LIN {X 0,Y 410.534,Z 444.335,A -85,B 0,C 180,E1 -10511.019,E2 -10511.019} C_VEL
LIN {X 0,Y 410.459,Z 447.37,A -85,B 0,C 180,E1 -10512.291,E2 -10512.291} C_VEL
LIN {X 0,Y 412.843,Z 460.26,A -85,B 0,C 180,E1 -10512.809,E2 -10512.809} C_VEL
LIN {X 0,Y 414.455,Z 473.213,A -85,B 0,C 180,E1 -10513.499,E2 -10513.499} C_VEL
LIN {X 0,Y 414.8,Z 477.532,A -85,B 0,C 180,E1 -10513.766,E2 -10513.766} C_VEL
LIN {X 0,Y 413.981,Z 489.912,A -85,B 0,C 180,E1 -10514.618,E2 -10514.618} C_VEL
LIN {X 0,Y 413.13,Z 501.048,A -85,B 0,C 180,E1 -10515.595,E2 -10515.595} C_VEL
LIN {X 0,Y 412.456,Z 511.121,A -85,B 0,C 180,E1 -10516.702,E2 -10516.702} C_VEL
LIN {X 0,Y 411.795,Z 520.263,A -85,B 0,C 180,E1 -10517.933,E2 -10517.933} C_VEL
LIN {X 0,Y 411.029,Z 529.203,A -85,B 0,C 180,E1 -10519.409,E2 -10519.409} C_VEL
LIN {X 0,Y 410.57,Z 536.417,A -85,B 0,C 180,E1 -10520.89,E2 -10520.89} C_VEL
LIN {X 0,Y 410.293,Z 541.303,A -85,B 0,C 180,E1 -10522.124,E2 -10522.124} C_VEL
LIN {X 0,Y 410.077,Z 546.418,A -85,B 0,C 180,E1 -10523.731,E2 -10523.731} C_VEL
LIN {X 0,Y 410.023,Z 549.684,A -85,B 0,C 180,E1 -10525.084,E2 -10525.084} C_VEL
LIN {X 0,Y 409.937,Z 551.546,A -85,B 0,C 180,E1 -10526.068,E2 -10526.068} C_VEL
LIN {X 0,Y 409.997,Z 553.956,A -85,B 0,C 180,E1 -10528.036,E2 -10528.036} C_VEL
LIN {X 0,Y 409.956,Z 554.566,A -85,B 0,C 180,E1 -10529.018,E2 -10529.018} C_VEL
LIN {X 0,Y 409.948,Z 554.761,A -85,B 0,C 180,E1 -10530,E2 -10530} C_VEL
LIN {X 0,Y 409.999,Z 553.907,A -85,B 0,C 180,E1 -10531.965,E2 -10531.965} C_VEL
LIN {X 0,Y 409.946,Z 552.887,A -85,B 0,C 180,E1 -10532.948,E2 -10532.948} C_VEL
LIN {X 0,Y 409.938,Z 551.437,A -85,B 0,C 180,E1 -10533.933,E2 -10533.933} C_VEL
LIN {X 0,Y 410.023,Z 548.439,A -85,B 0,C 180,E1 -10535.41,E2 -10535.41} C_VEL
LIN {X 0,Y 410.166,Z 544.376,A -85,B 0,C 180,E1 -10536.889,E2 -10536.889} C_VEL
LIN {X 0,Y 410.467,Z 538.12,A -85,B 0,C 180,E1 -10538.617,E2 -10538.617} C_VEL
LIN {X 0,Y 410.893,Z 531.306,A -85,B 0,C 180,E1 -10540.097,E2 -10540.097} C_VEL
LIN {X 0,Y 411.324,Z 524.356,A -85,B 0,C 180,E1 -10541.332,E2 -10541.332} C_VEL
LIN {X 0,Y 411.998,Z 515.999,A -85,B 0,C 180,E1 -10542.562,E2 -10542.562} C_VEL
LIN {X 0,Y 412.657,Z 505.728,A -85,B 0,C 180,E1 -10543.794,E2 -10543.794} C_VEL
LIN {X 0,Y 413.456,Z 494.162,A -85,B 0,C 180,E1 -10544.898,E2 -10544.898} C_VEL
LIN {X 0,Y 414.251,Z 482.81,A -85,B 0,C 180,E1 -10545.751,E2 -10545.751} C_VEL
LIN {X 0,Y 414.417,Z 475.557,A -85,B 0,C 180,E1 -10546.197,E2 -10546.197} C_VEL
LIN {X 0,Y 412.714,Z 461.921,A -85,B 0,C 180,E1 -10546.926,E2 -10546.926} C_VEL
LIN {X 0,Y 410.687,Z 449.667,A -85,B 0,C 180,E1 -10547.409,E2 -10547.409} C_VEL
LIN {X 0,Y 410.428,Z 447.964,A -85,B 0,C 180,E1 -10547.469,E2 -10547.469} C_VEL
LIN {X 0,Y 410.774,Z 440.007,A -85,B 0,C 180,E1 -10551.057,E2 -10551.057} C_VEL
LIN {X 0,Y 411.056,Z 433.097,A -85,B 0,C 180,E1 -10554.226,E2 -10554.226} C_VEL
LIN {X 0,Y 411.471,Z 426.207,A -85,B 0,C 180,E1 -10557.462,E2 -10557.462} C_VEL
LIN {X 0,Y 411.896,Z 420.472,A -85,B 0,C 180,E1 -10560.222,E2 -10560.222} C_VEL
LIN {X 0,Y 412.375,Z 414.103,A -85,B 0,C 180,E1 -10563.374,E2 -10563.374} C_VEL
LIN {X 0,Y 412.666,Z 410.157,A -85,B 0,C 180,E1 -10565.384,E2 -10565.384} C_VEL
LIN {X 0,Y 412.285,Z 405.559,A -85,B 0,C 180,E1 -10567.856,E2 -10567.856} C_VEL
LIN {X 0,Y 411.558,Z 400.956,A -85,B 0,C 180,E1 -10570.46,E2 -10570.46} C_VEL
LIN {X 0,Y 411.242,Z 399.261,A -85,B 0,C 180,E1 -10571.557,E2 -10571.557} C_VEL
LIN {X 0,Y 411.177,Z 399.269,A -85,B 0,C 180,E1 -10575.51,E2 -10575.51} C_VEL
LIN {X 0,Y 411.165,Z 399.27,A -85,B 0,C 180,E1 -10578.772,E2 -10578.772} C_VEL
LIN {X 0,Y 411.194,Z 399.264,A -85,B 0,C 180,E1 -10582.026,E2 -10582.026} C_VEL
LIN {X 0,Y 411.207,Z 399.263,A -85,B 0,C 180,E1 -10585.666,E2 -10585.666} C_VEL
LIN {X 0,Y 411.19,Z 399.268,A -85,B 0,C 180,E1 -10589.152,E2 -10589.152} C_VEL
LIN {X 0,Y 411.26,Z 399.256,A -85,B 0,C 180,E1 -10592.522,E2 -10592.522} C_VEL
LIN {X 0,Y 411.228,Z 399.261,A -85,B 0,C 180,E1 -10595.785,E2 -10595.785} C_VEL
LIN {X 0,Y 411.197,Z 399.267,A -85,B 0,C 180,E1 -10598.966,E2 -10598.966} C_VEL
LIN {X 0,Y 411.253,Z 399.257,A -85,B 0,C 180,E1 -10602.085,E2 -10602.085} C_VEL
LIN {X 0,Y 411.26,Z 399.259,A -85,B 0,C 180,E1 -10605.147,E2 -10605.147} C_VEL
LIN {X 0,Y 411.285,Z 399.253,A -85,B 0,C 180,E1 -10608.167,E2 -10608.167} C_VEL
LIN {X 0,Y 411.483,Z 399.228,A -85,B 0,C 180,E1 -10612.147,E2 -10612.147} C_VEL
LIN {X 0,Y 411.475,Z 399.229,A -85,B 0,C 180,E1 -10614.118,E2 -10614.118} C_VEL
LIN {X 0,Y 411.511,Z 399.224,A -85,B 0,C 180,E1 -10618.042,E2 -10618.042} C_VEL
LIN {X 0,Y 411.64,Z 399.208,A -85,B 0,C 180,E1 -10620,E2 -10620} C_VEL
LIN {X 0,Y 411.458,Z 399.234,A -85,B 0,C 180,E1 -10622.937,E2 -10622.937} C_VEL
LIN {X 0,Y 411.461,Z 399.234,A -85,B 0,C 180,E1 -10626.867,E2 -10626.867} C_VEL
LIN {X 0,Y 411.355,Z 399.247,A -85,B 0,C 180,E1 -10628.845,E2 -10628.845} C_VEL
LIN {X 0,Y 411.284,Z 399.253,A -85,B 0,C 180,E1 -10631.833,E2 -10631.833} C_VEL
LIN {X 0,Y 411.26,Z 399.259,A -85,B 0,C 180,E1 -10634.853,E2 -10634.853} C_VEL
LIN {X 0,Y 411.253,Z 399.257,A -85,B 0,C 180,E1 -10637.915,E2 -10637.915} C_VEL
LIN {X 0,Y 411.197,Z 399.267,A -85,B 0,C 180,E1 -10641.034,E2 -10641.034} C_VEL
LIN {X 0,Y 411.227,Z 399.261,A -85,B 0,C 180,E1 -10644.215,E2 -10644.215} C_VEL
LIN {X 0,Y 411.259,Z 399.256,A -85,B 0,C 180,E1 -10647.478,E2 -10647.478} C_VEL
LIN {X 0,Y 411.19,Z 399.268,A -85,B 0,C 180,E1 -10650.848,E2 -10650.848} C_VEL
LIN {X 0,Y 411.207,Z 399.264,A -85,B 0,C 180,E1 -10654.333,E2 -10654.333} C_VEL
LIN {X 0,Y 411.194,Z 399.264,A -85,B 0,C 180,E1 -10657.974,E2 -10657.974} C_VEL
LIN {X 0,Y 411.164,Z 399.269,A -85,B 0,C 180,E1 -10661.228,E2 -10661.228} C_VEL
LIN {X 0,Y 411.176,Z 399.27,A -85,B 0,C 180,E1 -10664.49,E2 -10664.49} C_VEL
LIN {X 0,Y 411.178,Z 399.269,A -85,B 0,C 180,E1 -10668.195,E2 -10668.195} C_VEL
LIN {X 0,Y 411.221,Z 399.264,A -85,B 0,C 180,E1 -10670.776,E2 -10670.776} C_VEL
LIN {X 0,Y 411.201,Z 399.266,A -85,B 0,C 180,E1 -10674.471,E2 -10674.471} C_VEL
LIN {X 0,Y 411.209,Z 399.265,A -85,B 0,C 180,E1 -10676.873,E2 -10676.873} C_VEL
LIN {X 0,Y 411.235,Z 399.263,A -85,B 0,C 180,E1 -10680.644,E2 -10680.644} C_VEL
LIN {X 0,Y 411.24,Z 399.258,A -85,B 0,C 180,E1 -10683.619,E2 -10683.619} C_VEL
LIN {X 0,Y 411.205,Z 399.264,A -85,B 0,C 180,E1 -10686.852,E2 -10686.852} C_VEL
LIN {X 0,Y 411.217,Z 399.263,A -85,B 0,C 180,E1 -10690.05,E2 -10690.05} C_VEL
LIN {X 0,Y 411.265,Z 399.255,A -85,B 0,C 180,E1 -10693.131,E2 -10693.131} C_VEL
LIN {X 0,Y 411.308,Z 399.251,A -85,B 0,C 180,E1 -10696.896,E2 -10696.896} C_VEL
LIN {X 0,Y 411.294,Z 399.255,A -85,B 0,C 180,E1 -10700.161,E2 -10700.161} C_VEL
LIN {X 0,Y 411.463,Z 399.231,A -85,B 0,C 180,E1 -10703.133,E2 -10703.133} C_VEL
LIN {X 0,Y 411.311,Z 399.249,A -85,B 0,C 180,E1 -10705.099,E2 -10705.099} C_VEL
LIN {X 0,Y 411.513,Z 399.227,A -85,B 0,C 180,E1 -10708.042,E2 -10708.042} C_VEL
LIN {X 0,Y 411.642,Z 399.211,A -85,B 0,C 180,E1 -10710,E2 -10710} C_VEL
LIN {X 0,Y 411.467,Z 399.231,A -85,B 0,C 180,E1 -10712.937,E2 -10712.937} C_VEL
LIN {X 0,Y 411.425,Z 399.238,A -85,B 0,C 180,E1 -10715.882,E2 -10715.882} C_VEL
LIN {X 0,Y 411.055,Z 399.284,A -85,B 0,C 180,E1 -10718.851,E2 -10718.851} C_VEL
LIN {X 0,Y 410.931,Z 399.893,A -85,B 0,C 180,E1 -10719.847,E2 -10719.847} C_VEL
LIN {X 0,Y 410.765,Z 403.877,A -85,B 0,C 180,E1 -10723.219,E2 -10723.219} C_VEL
LIN {X 0,Y 410.587,Z 407.911,A -85,B 0,C 180,E1 -10726.554,E2 -10726.554} C_VEL
LIN {X 0,Y 410.492,Z 408.997,A -85,B 0,C 180,E1 -10727.431,E2 -10727.431} C_VEL
LIN {X 0,Y 409.759,Z 410.069,A -85,B 0,C 180,E1 -10728.236,E2 -10728.236} C_VEL
LIN {X 0,Y 406.821,Z 411.984,A -85,B 0,C 180,E1 -10729.538,E2 -10729.538} C_VEL
LIN {X 0,Y 404.358,Z 413.528,A -85,B 0,C 180,E1 -10730.59,E2 -10730.59} C_VEL
LIN {X 0,Y 403.295,Z 414.632,A -85,B 0,C 180,E1 -10731.405,E2 -10731.405} C_VEL
LIN {X 0,Y 403.204,Z 414.98,A -85,B 0,C 180,E1 -10731.683,E2 -10731.683} C_VEL
LIN {X 0,Y 403.126,Z 419.403,A -85,B 0,C 180,E1 -10735.224,E2 -10735.224} C_VEL
LIN {X 0,Y 403.12,Z 419.529,A -85,B 0,C 180,E1 -10735.323,E2 -10735.323} C_VEL
LIN {X 0,Y 406.742,Z 435.397,A -85,B 0,C 180,E1 -10736.073,E2 -10736.073} C_VEL
LIN {X 0,Y 408.218,Z 444.133,A -85,B 0,C 180,E1 -10736.591,E2 -10736.591} C_VEL
LIN {X 0,Y 407.522,Z 455.702,A -85,B 0,C 180,E1 -10737.333,E2 -10737.333} C_VEL
LIN {X 0,Y 406.846,Z 466.667,A -85,B 0,C 180,E1 -10738.238,E2 -10738.238} C_VEL
LIN {X 0,Y 406.077,Z 477.882,A -85,B 0,C 180,E1 -10739.411,E2 -10739.411} C_VEL
LIN {X 0,Y 405.377,Z 487.193,A -85,B 0,C 180,E1 -10740.615,E2 -10740.615} C_VEL
LIN {X 0,Y 404.747,Z 495.157,A -85,B 0,C 180,E1 -10741.866,E2 -10741.866} C_VEL
LIN {X 0,Y 404.142,Z 503.143,A -85,B 0,C 180,E1 -10743.414,E2 -10743.414} C_VEL
LIN {X 0,Y 403.603,Z 509.906,A -85,B 0,C 180,E1 -10745.073,E2 -10745.073} C_VEL
LIN {X 0,Y 403.245,Z 515.072,A -85,B 0,C 180,E1 -10746.706,E2 -10746.706} C_VEL
LIN {X 0,Y 403.02,Z 518.865,A -85,B 0,C 180,E1 -10748.305,E2 -10748.305} C_VEL
LIN {X 0,Y 402.771,Z 521.882,A -85,B 0,C 180,E1 -10750.211,E2 -10750.211} C_VEL
LIN {X 0,Y 402.72,Z 523.128,A -85,B 0,C 180,E1 -10751.54,E2 -10751.54} C_VEL
LIN {X 0,Y 402.728,Z 523.627,A -85,B 0,C 180,E1 -10752.889,E2 -10752.889} C_VEL
LIN {X 0,Y 402.74,Z 523.385,A -85,B 0,C 180,E1 -10754.318,E2 -10754.318} C_VEL
LIN {X 0,Y 402.808,Z 522.35,A -85,B 0,C 180,E1 -10755.741,E2 -10755.741} C_VEL
LIN {X 0,Y 402.952,Z 520.541,A -85,B 0,C 180,E1 -10757.14,E2 -10757.14} C_VEL
LIN {X 0,Y 403.182,Z 517.849,A -85,B 0,C 180,E1 -10758.55,E2 -10758.55} C_VEL
LIN {X 0,Y 403.438,Z 514.039,A -85,B 0,C 180,E1 -10760.039,E2 -10760.039} C_VEL
LIN {X 0,Y 403.834,Z 509.049,A -85,B 0,C 180,E1 -10761.548,E2 -10761.548} C_VEL
LIN {X 0,Y 404.367,Z 502.647,A -85,B 0,C 180,E1 -10763.08,E2 -10763.08} C_VEL
LIN {X 0,Y 405.072,Z 494.485,A -85,B 0,C 180,E1 -10764.631,E2 -10764.631} C_VEL
LIN {X 0,Y 405.853,Z 485.639,A -85,B 0,C 180,E1 -10765.988,E2 -10765.988} C_VEL
LIN {X 0,Y 406.63,Z 476.25,A -85,B 0,C 180,E1 -10767.162,E2 -10767.162} C_VEL
LIN {X 0,Y 407.461,Z 465.3,A -85,B 0,C 180,E1 -10768.259,E2 -10768.259} C_VEL
LIN {X 0,Y 408.228,Z 453.199,A -85,B 0,C 180,E1 -10769.22,E2 -10769.22} C_VEL
LIN {X 0,Y 408.72,Z 443.775,A -85,B 0,C 180,E1 -10769.804,E2 -10769.804} C_VEL
LIN {X 0,Y 406.173,Z 431.616,A -85,B 0,C 180,E1 -10770.537,E2 -10770.537} C_VEL
LIN {X 0,Y 403.286,Z 420.513,A -85,B 0,C 180,E1 -10771.08,E2 -10771.08} C_VEL
LIN {X 0,Y 403.395,Z 416.813,A -85,B 0,C 180,E1 -10774.179,E2 -10774.179} C_VEL
LIN {X 0,Y 403.589,Z 412.981,A -85,B 0,C 180,E1 -10777.474,E2 -10777.474} C_VEL
LIN {X 0,Y 403.803,Z 409.322,A -85,B 0,C 180,E1 -10780.69,E2 -10780.69} C_VEL
LIN {X 0,Y 404.001,Z 405.837,A -85,B 0,C 180,E1 -10783.839,E2 -10783.839} C_VEL
LIN {X 0,Y 404.23,Z 402.512,A -85,B 0,C 180,E1 -10786.937,E2 -10786.937} C_VEL
LIN {X 0,Y 404.177,Z 400.432,A -85,B 0,C 180,E1 -10788.973,E2 -10788.973} C_VEL
LIN {X 0,Y 404.281,Z 400.133,A -85,B 0,C 180,E1 -10790.999,E2 -10790.999} C_VEL
LIN {X 0,Y 404.407,Z 400.113,A -85,B 0,C 180,E1 -10793.013,E2 -10793.013} C_VEL
LIN {X 0,Y 404.28,Z 400.129,A -85,B 0,C 180,E1 -10795.014,E2 -10795.014} C_VEL
LIN {X 0,Y 404.479,Z 400.105,A -85,B 0,C 180,E1 -10798.009,E2 -10798.009} C_VEL
LIN {X 0,Y 404.609,Z 400.087,A -85,B 0,C 180,E1 -10800,E2 -10800} C_VEL
LIN {X 0,Y 404.419,Z 400.112,A -85,B 0,C 180,E1 -10802.988,E2 -10802.988} C_VEL
LIN {X 0,Y 404.408,Z 400.113,A -85,B 0,C 180,E1 -10806.987,E2 -10806.987} C_VEL
LIN {X 0,Y 404.254,Z 400.132,A -85,B 0,C 180,E1 -10810.012,E2 -10810.012} C_VEL
LIN {X 0,Y 404.262,Z 400.131,A -85,B 0,C 180,E1 -10813.212,E2 -10813.212} C_VEL
LIN {X 0,Y 404.212,Z 400.137,A -85,B 0,C 180,E1 -10817.007,E2 -10817.007} C_VEL
LIN {X 0,Y 404.16,Z 400.143,A -85,B 0,C 180,E1 -10820.352,E2 -10820.352} C_VEL
LIN {X 0,Y 404.166,Z 400.141,A -85,B 0,C 180,E1 -10823.575,E2 -10823.575} C_VEL
LIN {X 0,Y 404.18,Z 400.141,A -85,B 0,C 180,E1 -10825.767,E2 -10825.767} C_VEL
LIN {X 0,Y 404.195,Z 400.139,A -85,B 0,C 180,E1 -10828,E2 -10828} C_VEL
LIN {X 0,Y 404.14,Z 400.146,A -85,B 0,C 180,E1 -10831.559,E2 -10831.559} C_VEL
LIN {X 0,Y 404.183,Z 400.143,A -85,B 0,C 180,E1 -10835.017,E2 -10835.017} C_VEL
LIN {X 0,Y 404.162,Z 400.145,A -85,B 0,C 180,E1 -10838.756,E2 -10838.756} C_VEL
LIN {X 0,Y 404.148,Z 400.147,A -85,B 0,C 180,E1 -10841.605,E2 -10841.605} C_VEL
LIN {X 0,Y 404.143,Z 400.147,A -85,B 0,C 180,E1 -10844.523,E2 -10844.523} C_VEL
LIN {X 0,Y 404.182,Z 400.333,A -85,B 0,C 180,E1 -10847.111,E2 -10847.111} C_VEL
LIN {X 0,Y 404.952,Z 404.545,A -85,B 0,C 180,E1 -10850.049,E2 -10850.049} C_VEL
LIN {X 0,Y 405.612,Z 408.992,A -85,B 0,C 180,E1 -10852.848,E2 -10852.848} C_VEL
LIN {X 0,Y 405.693,Z 412.911,A -85,B 0,C 180,E1 -10855.134,E2 -10855.134} C_VEL
LIN {X 0,Y 405.279,Z 417.229,A -85,B 0,C 180,E1 -10857.482,E2 -10857.482} C_VEL
LIN {X 0,Y 404.815,Z 422.492,A -85,B 0,C 180,E1 -10860.233,E2 -10860.233} C_VEL
LIN {X 0,Y 404.277,Z 429.369,A -85,B 0,C 180,E1 -10863.686,E2 -10863.686} C_VEL
LIN {X 0,Y 403.856,Z 437.27,A -85,B 0,C 180,E1 -10867.49,E2 -10867.49} C_VEL
LIN {X 0,Y 403.467,Z 444.131,A -85,B 0,C 180,E1 -10870.673,E2 -10870.673} C_VEL
LIN {X 0,Y 403.404,Z 447.055,A -85,B 0,C 180,E1 -10871.938,E2 -10871.938} C_VEL
LIN {X 0,Y 405.856,Z 459.934,A -85,B 0,C 180,E1 -10872.478,E2 -10872.478} C_VEL
LIN {X 0,Y 407.465,Z 472.667,A -85,B 0,C 180,E1 -10873.171,E2 -10873.171} C_VEL
LIN {X 0,Y 407.878,Z 479.72,A -85,B 0,C 180,E1 -10873.625,E2 -10873.625} C_VEL
LIN {X 0,Y 407.042,Z 491.446,A -85,B 0,C 180,E1 -10874.478,E2 -10874.478} C_VEL
LIN {X 0,Y 406.123,Z 502.634,A -85,B 0,C 180,E1 -10875.52,E2 -10875.52} C_VEL
LIN {X 0,Y 405.407,Z 513.072,A -85,B 0,C 180,E1 -10876.737,E2 -10876.737} C_VEL
LIN {X 0,Y 404.665,Z 521.747,A -85,B 0,C 180,E1 -10877.971,E2 -10877.971} C_VEL
LIN {X 0,Y 403.927,Z 530.331,A -85,B 0,C 180,E1 -10879.474,E2 -10879.474} C_VEL
LIN {X 0,Y 403.482,Z 537.235,A -85,B 0,C 180,E1 -10880.981,E2 -10880.981} C_VEL
LIN {X 0,Y 403.14,Z 542.775,A -85,B 0,C 180,E1 -10882.488,E2 -10882.488} C_VEL
LIN {X 0,Y 402.946,Z 547.124,A -85,B 0,C 180,E1 -10883.993,E2 -10883.993} C_VEL
LIN {X 0,Y 402.935,Z 549.437,A -85,B 0,C 180,E1 -10884.997,E2 -10884.997} C_VEL
LIN {X 0,Y 402.857,Z 551.29,A -85,B 0,C 180,E1 -10885.999,E2 -10885.999} C_VEL
LIN {X 0,Y 402.907,Z 553.694,A -85,B 0,C 180,E1 -10888.001,E2 -10888.001} C_VEL
LIN {X 0,Y 402.882,Z 554.301,A -85,B 0,C 180,E1 -10889.001,E2 -10889.001} C_VEL
LIN {X 0,Y 402.871,Z 554.486,A -85,B 0,C 180,E1 -10890,E2 -10890} C_VEL
LIN {X 0,Y 402.882,Z 554.249,A -85,B 0,C 180,E1 -10891,E2 -10891} C_VEL
LIN {X 0,Y 402.909,Z 553.622,A -85,B 0,C 180,E1 -10892,E2 -10892} C_VEL
LIN {X 0,Y 402.846,Z 552.596,A -85,B 0,C 180,E1 -10893,E2 -10893} C_VEL
LIN {X 0,Y 402.859,Z 551.134,A -85,B 0,C 180,E1 -10894.002,E2 -10894.002} C_VEL
LIN {X 0,Y 402.924,Z 548.124,A -85,B 0,C 180,E1 -10895.505,E2 -10895.505} C_VEL
LIN {X 0,Y 403.078,Z 544.046,A -85,B 0,C 180,E1 -10897.011,E2 -10897.011} C_VEL
LIN {X 0,Y 403.404,Z 537.772,A -85,B 0,C 180,E1 -10898.769,E2 -10898.769} C_VEL
LIN {X 0,Y 403.838,Z 530.939,A -85,B 0,C 180,E1 -10900.276,E2 -10900.276} C_VEL
LIN {X 0,Y 404.346,Z 523.971,A -85,B 0,C 180,E1 -10901.53,E2 -10901.53} C_VEL
LIN {X 0,Y 405.021,Z 515.589,A -85,B 0,C 180,E1 -10902.782,E2 -10902.782} C_VEL
LIN {X 0,Y 405.721,Z 505.059,A -85,B 0,C 180,E1 -10904.058,E2 -10904.058} C_VEL
LIN {X 0,Y 406.57,Z 493.673,A -85,B 0,C 180,E1 -10905.157,E2 -10905.157} C_VEL
LIN {X 0,Y 407.378,Z 482.257,A -85,B 0,C 180,E1 -10906.024,E2 -10906.024} C_VEL
LIN {X 0,Y 407.429,Z 475.56,A -85,B 0,C 180,E1 -10906.446,E2 -10906.446} C_VEL
LIN {X 0,Y 405.74,Z 462.081,A -85,B 0,C 180,E1 -10907.184,E2 -10907.184} C_VEL
LIN {X 0,Y 403.629,Z 449.579,A -85,B 0,C 180,E1 -10907.692,E2 -10907.692} C_VEL
LIN {X 0,Y 403.376,Z 447.773,A -85,B 0,C 180,E1 -10907.748,E2 -10907.748} C_VEL
LIN {X 0,Y 403.673,Z 440.877,A -85,B 0,C 180,E1 -10910.911,E2 -10910.911} C_VEL
LIN {X 0,Y 403.978,Z 433.991,A -85,B 0,C 180,E1 -10914.132,E2 -10914.132} C_VEL
LIN {X 0,Y 404.44,Z 426.747,A -85,B 0,C 180,E1 -10917.596,E2 -10917.596} C_VEL
LIN {X 0,Y 404.956,Z 420.241,A -85,B 0,C 180,E1 -10920.795,E2 -10920.795} C_VEL
LIN {X 0,Y 405.516,Z 413.356,A -85,B 0,C 180,E1 -10924.282,E2 -10924.282} C_VEL
LIN {X 0,Y 405.607,Z 409.937,A -85,B 0,C 180,E1 -10926.095,E2 -10926.095} C_VEL
LIN {X 0,Y 405.092,Z 405.284,A -85,B 0,C 180,E1 -10928.674,E2 -10928.674} C_VEL
LIN {X 0,Y 404.175,Z 400.141,A -85,B 0,C 180,E1 -10931.713,E2 -10931.713} C_VEL
LIN {X 0,Y 404.147,Z 400.145,A -85,B 0,C 180,E1 -10935.478,E2 -10935.478} C_VEL
LIN {X 0,Y 404.119,Z 400.146,A -85,B 0,C 180,E1 -10938.635,E2 -10938.635} C_VEL
LIN {X 0,Y 404.153,Z 400.144,A -85,B 0,C 180,E1 -10941.492,E2 -10941.492} C_VEL
LIN {X 0,Y 404.186,Z 400.14,A -85,B 0,C 180,E1 -10944.984,E2 -10944.984} C_VEL
LIN {X 0,Y 404.143,Z 400.143,A -85,B 0,C 180,E1 -10948.554,E2 -10948.554} C_VEL
LIN {X 0,Y 404.196,Z 400.135,A -85,B 0,C 180,E1 -10952,E2 -10952} C_VEL
LIN {X 0,Y 404.178,Z 400.141,A -85,B 0,C 180,E1 -10955.334,E2 -10955.334} C_VEL
LIN {X 0,Y 404.139,Z 400.144,A -85,B 0,C 180,E1 -10958.581,E2 -10958.581} C_VEL
LIN {X 0,Y 404.211,Z 400.134,A -85,B 0,C 180,E1 -10961.762,E2 -10961.762} C_VEL
LIN {X 0,Y 404.207,Z 400.138,A -85,B 0,C 180,E1 -10964.882,E2 -10964.882} C_VEL
LIN {X 0,Y 404.257,Z 400.128,A -85,B 0,C 180,E1 -10967.958,E2 -10967.958} C_VEL
LIN {X 0,Y 404.434,Z 400.106,A -85,B 0,C 180,E1 -10972.1,E2 -10972.1} C_VEL
LIN {X 0,Y 404.424,Z 400.107,A -85,B 0,C 180,E1 -10974.015,E2 -10974.015} C_VEL
LIN {X 0,Y 404.48,Z 400.1,A -85,B 0,C 180,E1 -10978.008,E2 -10978.008} C_VEL
LIN {X 0,Y 404.61,Z 400.084,A -85,B 0,C 180,E1 -10980,E2 -10980} C_VEL
LIN {X 0,Y 404.416,Z 400.111,A -85,B 0,C 180,E1 -10982.988,E2 -10982.988} C_VEL
LIN {X 0,Y 404.412,Z 400.113,A -85,B 0,C 180,E1 -10986.987,E2 -10986.987} C_VEL
LIN {X 0,Y 404.259,Z 400.128,A -85,B 0,C 180,E1 -10990.012,E2 -10990.012} C_VEL
LIN {X 0,Y 404.267,Z 400.129,A -85,B 0,C 180,E1 -10993.211,E2 -10993.211} C_VEL
LIN {X 0,Y 404.216,Z 400.136,A -85,B 0,C 180,E1 -10997.007,E2 -10997.007} C_VEL
LIN {X 0,Y 404.164,Z 400.141,A -85,B 0,C 180,E1 -11000.352,E2 -11000.352} C_VEL
LIN {X 0,Y 404.17,Z 400.139,A -85,B 0,C 180,E1 -11003.574,E2 -11003.574} C_VEL
LIN {X 0,Y 404.184,Z 400.136,A -85,B 0,C 180,E1 -11005.766,E2 -11005.766} C_VEL
LIN {X 0,Y 404.196,Z 400.136,A -85,B 0,C 180,E1 -11008,E2 -11008} C_VEL
LIN {X 0,Y 404.14,Z 400.142,A -85,B 0,C 180,E1 -11011.558,E2 -11011.558} C_VEL
LIN {X 0,Y 404.186,Z 400.139,A -85,B 0,C 180,E1 -11015.016,E2 -11015.016} C_VEL
LIN {X 0,Y 404.153,Z 400.144,A -85,B 0,C 180,E1 -11018.757,E2 -11018.757} C_VEL
LIN {X 0,Y 404.123,Z 400.145,A -85,B 0,C 180,E1 -11021.6,E2 -11021.6} C_VEL
LIN {X 0,Y 404.146,Z 400.145,A -85,B 0,C 180,E1 -11024.522,E2 -11024.522} C_VEL
LIN {X 0,Y 404.137,Z 400.143,A -85,B 0,C 180,E1 -11027.296,E2 -11027.296} C_VEL
LIN {X 0,Y 404.17,Z 400.139,A -85,B 0,C 180,E1 -11029.955,E2 -11029.955} C_VEL
LIN {X 0,Y 404.141,Z 400.144,A -85,B 0,C 180,E1 -11033.124,E2 -11033.124} C_VEL
LIN {X 0,Y 404.146,Z 400.144,A -85,B 0,C 180,E1 -11036.188,E2 -11036.188} C_VEL
LIN {X 0,Y 404.147,Z 400.142,A -85,B 0,C 180,E1 -11039.715,E2 -11039.715} C_VEL
LIN {X 0,Y 404.197,Z 400.136,A -85,B 0,C 180,E1 -11043.123,E2 -11043.123} C_VEL
LIN {X 0,Y 404.179,Z 400.138,A -85,B 0,C 180,E1 -11045.334,E2 -11045.334} C_VEL
LIN {X 0,Y 404.141,Z 400.146,A -85,B 0,C 180,E1 -11048.581,E2 -11048.581} C_VEL
LIN {X 0,Y 404.212,Z 400.134,A -85,B 0,C 180,E1 -11051.762,E2 -11051.762} C_VEL
LIN {X 0,Y 404.208,Z 400.136,A -85,B 0,C 180,E1 -11054.882,E2 -11054.882} C_VEL
LIN {X 0,Y 404.258,Z 400.13,A -85,B 0,C 180,E1 -11057.958,E2 -11057.958} C_VEL
LIN {X 0,Y 404.436,Z 400.108,A -85,B 0,C 180,E1 -11062.099,E2 -11062.099} C_VEL
LIN {X 0,Y 404.426,Z 400.11,A -85,B 0,C 180,E1 -11064.015,E2 -11064.015} C_VEL
LIN {X 0,Y 404.482,Z 400.102,A -85,B 0,C 180,E1 -11068.008,E2 -11068.008} C_VEL
LIN {X 0,Y 404.612,Z 400.087,A -85,B 0,C 180,E1 -11070,E2 -11070} C_VEL
LIN {X 0,Y 404.424,Z 400.108,A -85,B 0,C 180,E1 -11072.988,E2 -11072.988} C_VEL
LIN {X 0,Y 404.368,Z 400.117,A -85,B 0,C 180,E1 -11075.985,E2 -11075.985} C_VEL
LIN {X 0,Y 403.984,Z 400.165,A -85,B 0,C 180,E1 -11079.007,E2 -11079.007} C_VEL
LIN {X 0,Y 403.862,Z 400.935,A -85,B 0,C 180,E1 -11080.021,E2 -11080.021} C_VEL
LIN {X 0,Y 403.743,Z 404.494,A -85,B 0,C 180,E1 -11083.078,E2 -11083.078} C_VEL
LIN {X 0,Y 403.521,Z 408.816,A -85,B 0,C 180,E1 -11086.681,E2 -11086.681} C_VEL
LIN {X 0,Y 403.276,Z 413.4,A -85,B 0,C 180,E1 -11090.398,E2 -11090.398} C_VEL
LIN {X 0,Y 403.204,Z 414.98,A -85,B 0,C 180,E1 -11091.683,E2 -11091.683} C_VEL
LIN {X 0,Y 402.505,Z 415.721,A -85,B 0,C 180,E1 -11092.229,E2 -11092.229} C_VEL
LIN {X 0,Y 399.618,Z 417.05,A -85,B 0,C 180,E1 -11093.078,E2 -11093.078} C_VEL
LIN {X 0,Y 396.74,Z 418.386,A -85,B 0,C 180,E1 -11093.938,E2 -11093.938} C_VEL
LIN {X 0,Y 396.079,Z 419.139,A -85,B 0,C 180,E1 -11094.497,E2 -11094.497} C_VEL
LIN {X 0,Y 396.082,Z 419.813,A -85,B 0,C 180,E1 -11095.041,E2 -11095.041} C_VEL
LIN {X 0,Y 399.357,Z 434.224,A -85,B 0,C 180,E1 -11095.715,E2 -11095.715} C_VEL
LIN {X 0,Y 401.345,Z 445.277,A -85,B 0,C 180,E1 -11096.381,E2 -11096.381} C_VEL
LIN {X 0,Y 400.627,Z 456.648,A -85,B 0,C 180,E1 -11097.135,E2 -11097.135} C_VEL
LIN {X 0,Y 399.91,Z 467.292,A -85,B 0,C 180,E1 -11098.04,E2 -11098.04} C_VEL
LIN {X 0,Y 399.092,Z 478.629,A -85,B 0,C 180,E1 -11099.256,E2 -11099.256} C_VEL
LIN {X 0,Y 398.284,Z 488.808,A -85,B 0,C 180,E1 -11100.619,E2 -11100.619} C_VEL
LIN {X 0,Y 397.593,Z 497.229,A -85,B 0,C 180,E1 -11102.024,E2 -11102.024} C_VEL
LIN {X 0,Y 396.954,Z 505.221,A -85,B 0,C 180,E1 -11103.682,E2 -11103.682} C_VEL
LIN {X 0,Y 396.455,Z 511.588,A -85,B 0,C 180,E1 -11105.368,E2 -11105.368} C_VEL
LIN {X 0,Y 396.116,Z 516.57,A -85,B 0,C 180,E1 -11107.101,E2 -11107.101} C_VEL
LIN {X 0,Y 395.882,Z 519.848,A -85,B 0,C 180,E1 -11108.637,E2 -11108.637} C_VEL
LIN {X 0,Y 395.689,Z 522.173,A -85,B 0,C 180,E1 -11110.205,E2 -11110.205} C_VEL
LIN {X 0,Y 395.641,Z 523.508,A -85,B 0,C 180,E1 -11111.749,E2 -11111.749} C_VEL
LIN {X 0,Y 395.643,Z 523.932,A -85,B 0,C 180,E1 -11113.256,E2 -11113.256} C_VEL
LIN {X 0,Y 395.675,Z 523.104,A -85,B 0,C 180,E1 -11115.273,E2 -11115.273} C_VEL
LIN {X 0,Y 395.801,Z 521.553,A -85,B 0,C 180,E1 -11116.719,E2 -11116.719} C_VEL
LIN {X 0,Y 396.047,Z 519.129,A -85,B 0,C 180,E1 -11118.184,E2 -11118.184} C_VEL
LIN {X 0,Y 396.297,Z 515.685,A -85,B 0,C 180,E1 -11119.69,E2 -11119.69} C_VEL
LIN {X 0,Y 396.676,Z 511.092,A -85,B 0,C 180,E1 -11121.219,E2 -11121.219} C_VEL
LIN {X 0,Y 397.282,Z 504.061,A -85,B 0,C 180,E1 -11123.025,E2 -11123.025} C_VEL
LIN {X 0,Y 398.029,Z 495.82,A -85,B 0,C 180,E1 -11124.675,E2 -11124.675} C_VEL
LIN {X 0,Y 398.789,Z 487.425,A -85,B 0,C 180,E1 -11126.021,E2 -11126.021} C_VEL
LIN {X 0,Y 399.774,Z 476.785,A -85,B 0,C 180,E1 -11127.403,E2 -11127.403} C_VEL
LIN {X 0,Y 400.63,Z 466.306,A -85,B 0,C 180,E1 -11128.484,E2 -11128.484} C_VEL
LIN {X 0,Y 401.447,Z 454.004,A -85,B 0,C 180,E1 -11129.49,E2 -11129.49} C_VEL
LIN {X 0,Y 402.01,Z 445.718,A -85,B 0,C 180,E1 -11130.022,E2 -11130.022} C_VEL
LIN {X 0,Y 399.721,Z 434.053,A -85,B 0,C 180,E1 -11130.761,E2 -11130.761} C_VEL
LIN {X 0,Y 396.256,Z 420.786,A -85,B 0,C 180,E1 -11131.468,E2 -11131.468} C_VEL
LIN {X 0,Y 396.404,Z 416.875,A -85,B 0,C 180,E1 -11134.817,E2 -11134.817} C_VEL
LIN {X 0,Y 396.564,Z 413.064,A -85,B 0,C 180,E1 -11138.151,E2 -11138.151} C_VEL
LIN {X 0,Y 396.789,Z 409.453,A -85,B 0,C 180,E1 -11141.408,E2 -11141.408} C_VEL
LIN {X 0,Y 397.002,Z 406.008,A -85,B 0,C 180,E1 -11144.601,E2 -11144.601} C_VEL
LIN {X 0,Y 397.196,Z 402.737,A -85,B 0,C 180,E1 -11147.741,E2 -11147.741} C_VEL
LIN {X 0,Y 397.162,Z 401.019,A -85,B 0,C 180,E1 -11149.808,E2 -11149.808} C_VEL
LIN {X 0,Y 397.39,Z 400.989,A -85,B 0,C 180,E1 -11152.041,E2 -11152.041} C_VEL
LIN {X 0,Y 397.252,Z 401.004,A -85,B 0,C 180,E1 -11154.925,E2 -11154.925} C_VEL
LIN {X 0,Y 397.448,Z 400.981,A -85,B 0,C 180,E1 -11157.973,E2 -11157.973} C_VEL
LIN {X 0,Y 397.578,Z 400.963,A -85,B 0,C 180,E1 -11160,E2 -11160} C_VEL
LIN {X 0,Y 397.377,Z 400.989,A -85,B 0,C 180,E1 -11163.041,E2 -11163.041} C_VEL
LIN {X 0,Y 397.36,Z 400.991,A -85,B 0,C 180,E1 -11167.112,E2 -11167.112} C_VEL
LIN {X 0,Y 397.214,Z 401.009,A -85,B 0,C 180,E1 -11170.191,E2 -11170.191} C_VEL
LIN {X 0,Y 397.222,Z 401.007,A -85,B 0,C 180,E1 -11173.321,E2 -11173.321} C_VEL
LIN {X 0,Y 397.178,Z 401.013,A -85,B 0,C 180,E1 -11177.155,E2 -11177.155} C_VEL
LIN {X 0,Y 397.099,Z 401.022,A -85,B 0,C 180,E1 -11180.73,E2 -11180.73} C_VEL
LIN {X 0,Y 397.129,Z 401.016,A -85,B 0,C 180,E1 -11184.019,E2 -11184.019} C_VEL
LIN {X 0,Y 397.191,Z 401.011,A -85,B 0,C 180,E1 -11187.391,E2 -11187.391} C_VEL
LIN {X 0,Y 397.082,Z 401.026,A -85,B 0,C 180,E1 -11190.882,E2 -11190.882} C_VEL
LIN {X 0,Y 397.123,Z 401.02,A -85,B 0,C 180,E1 -11194.494,E2 -11194.494} C_VEL
LIN {X 0,Y 397.108,Z 401.024,A -85,B 0,C 180,E1 -11198.275,E2 -11198.275} C_VEL
LIN {X 0,Y 397.111,Z 401.023,A -85,B 0,C 180,E1 -11200.906,E2 -11200.906} C_VEL
LIN {X 0,Y 397.1,Z 401.024,A -85,B 0,C 180,E1 -11203.649,E2 -11203.649} C_VEL
LIN {X 0,Y 397.148,Z 401.216,A -85,B 0,C 180,E1 -11206.699,E2 -11206.699} C_VEL
LIN {X 0,Y 397.824,Z 405.035,A -85,B 0,C 180,E1 -11209.433,E2 -11209.433} C_VEL
LIN {X 0,Y 398.545,Z 409.725,A -85,B 0,C 180,E1 -11212.518,E2 -11212.518} C_VEL
LIN {X 0,Y 398.742,Z 412.909,A -85,B 0,C 180,E1 -11214.435,E2 -11214.435} C_VEL
LIN {X 0,Y 398.348,Z 417.163,A -85,B 0,C 180,E1 -11216.844,E2 -11216.844} C_VEL
LIN {X 0,Y 397.83,Z 422.941,A -85,B 0,C 180,E1 -11219.955,E2 -11219.955} C_VEL
LIN {X 0,Y 397.22,Z 430.344,A -85,B 0,C 180,E1 -11223.748,E2 -11223.748} C_VEL
LIN {X 0,Y 396.836,Z 437.105,A -85,B 0,C 180,E1 -11227.07,E2 -11227.07} C_VEL
LIN {X 0,Y 396.438,Z 443.913,A -85,B 0,C 180,E1 -11230.317,E2 -11230.317} C_VEL
LIN {X 0,Y 396.324,Z 446.553,A -85,B 0,C 180,E1 -11231.554,E2 -11231.554} C_VEL
LIN {X 0,Y 399.07,Z 460.698,A -85,B 0,C 180,E1 -11232.183,E2 -11232.183} C_VEL
LIN {X 0,Y 400.612,Z 473.302,A -85,B 0,C 180,E1 -11232.901,E2 -11232.901} C_VEL
LIN {X 0,Y 401.059,Z 479.993,A -85,B 0,C 180,E1 -11233.351,E2 -11233.351} C_VEL
LIN {X 0,Y 400.185,Z 491.419,A -85,B 0,C 180,E1 -11234.205,E2 -11234.205} C_VEL
LIN {X 0,Y 399.227,Z 502.535,A -85,B 0,C 180,E1 -11235.264,E2 -11235.264} C_VEL
LIN {X 0,Y 398.447,Z 513.138,A -85,B 0,C 180,E1 -11236.527,E2 -11236.527} C_VEL
LIN {X 0,Y 397.697,Z 521.593,A -85,B 0,C 180,E1 -11237.757,E2 -11237.757} C_VEL
LIN {X 0,Y 396.911,Z 530.146,A -85,B 0,C 180,E1 -11239.286,E2 -11239.286} C_VEL
LIN {X 0,Y 396.412,Z 537.035,A -85,B 0,C 180,E1 -11240.819,E2 -11240.819} C_VEL
LIN {X 0,Y 396.069,Z 542.562,A -85,B 0,C 180,E1 -11242.353,E2 -11242.353} C_VEL
LIN {X 0,Y 395.835,Z 547.638,A -85,B 0,C 180,E1 -11244.183,E2 -11244.183} C_VEL
LIN {X 0,Y 395.779,Z 551.044,A -85,B 0,C 180,E1 -11245.927,E2 -11245.927} C_VEL
LIN {X 0,Y 395.805,Z 553.435,A -85,B 0,C 180,E1 -11247.965,E2 -11247.965} C_VEL
LIN {X 0,Y 395.81,Z 554.038,A -85,B 0,C 180,E1 -11248.983,E2 -11248.983} C_VEL
LIN {X 0,Y 395.797,Z 554.21,A -85,B 0,C 180,E1 -11250,E2 -11250} C_VEL
LIN {X 0,Y 395.81,Z 553.968,A -85,B 0,C 180,E1 -11251.018,E2 -11251.018} C_VEL
LIN {X 0,Y 395.823,Z 553.335,A -85,B 0,C 180,E1 -11252.035,E2 -11252.035} C_VEL
LIN {X 0,Y 395.747,Z 552.303,A -85,B 0,C 180,E1 -11253.054,E2 -11253.054} C_VEL
LIN {X 0,Y 395.783,Z 550.828,A -85,B 0,C 180,E1 -11254.073,E2 -11254.073} C_VEL
LIN {X 0,Y 395.831,Z 547.295,A -85,B 0,C 180,E1 -11255.81,E2 -11255.81} C_VEL
LIN {X 0,Y 396.067,Z 542.077,A -85,B 0,C 180,E1 -11257.648,E2 -11257.648} C_VEL
LIN {X 0,Y 396.4,Z 536.393,A -85,B 0,C 180,E1 -11259.182,E2 -11259.182} C_VEL
LIN {X 0,Y 396.866,Z 529.255,A -85,B 0,C 180,E1 -11260.716,E2 -11260.716} C_VEL
LIN {X 0,Y 397.649,Z 520.366,A -85,B 0,C 180,E1 -11262.245,E2 -11262.245} C_VEL
LIN {X 0,Y 398.296,Z 511.648,A -85,B 0,C 180,E1 -11263.468,E2 -11263.468} C_VEL
LIN {X 0,Y 399.077,Z 501.195,A -85,B 0,C 180,E1 -11264.664,E2 -11264.664} C_VEL
LIN {X 0,Y 399.921,Z 490.058,A -85,B 0,C 180,E1 -11265.676,E2 -11265.676} C_VEL
LIN {X 0,Y 400.666,Z 478.604,A -85,B 0,C 180,E1 -11266.497,E2 -11266.497} C_VEL
LIN {X 0,Y 399.359,Z 466.306,A -85,B 0,C 180,E1 -11267.241,E2 -11267.241} C_VEL
LIN {X 0,Y 397.287,Z 453.084,A -85,B 0,C 180,E1 -11267.845,E2 -11267.845} C_VEL
LIN {X 0,Y 396.314,Z 447.476,A -85,B 0,C 180,E1 -11268.063,E2 -11268.063} C_VEL
LIN {X 0,Y 396.624,Z 440.591,A -85,B 0,C 180,E1 -11271.3,E2 -11271.3} C_VEL
LIN {X 0,Y 396.978,Z 433.715,A -85,B 0,C 180,E1 -11274.585,E2 -11274.585} C_VEL
LIN {X 0,Y 397.414,Z 427.049,A -85,B 0,C 180,E1 -11277.844,E2 -11277.844} C_VEL
LIN {X 0,Y 397.911,Z 421.135,A -85,B 0,C 180,E1 -11280.811,E2 -11280.811} C_VEL
LIN {X 0,Y 398.512,Z 414.28,A -85,B 0,C 180,E1 -11284.357,E2 -11284.357} C_VEL
LIN {X 0,Y 398.6,Z 411.586,A -85,B 0,C 180,E1 -11285.8,E2 -11285.8} C_VEL
LIN {X 0,Y 398.22,Z 407.393,A -85,B 0,C 180,E1 -11288.148,E2 -11288.148} C_VEL
LIN {X 0,Y 397.435,Z 402.797,A -85,B 0,C 180,E1 -11290.866,E2 -11290.866} C_VEL
LIN {X 0,Y 397.123,Z 401.02,A -85,B 0,C 180,E1 -11291.988,E2 -11291.988} C_VEL
LIN {X 0,Y 397.088,Z 401.025,A -85,B 0,C 180,E1 -11295.069,E2 -11295.069} C_VEL
LIN {X 0,Y 397.067,Z 401.024,A -85,B 0,C 180,E1 -11298.021,E2 -11298.021} C_VEL
LIN {X 0,Y 397.129,Z 401.019,A -85,B 0,C 180,E1 -11301.139,E2 -11301.139} C_VEL
LIN {X 0,Y 397.12,Z 401.017,A -85,B 0,C 180,E1 -11304.497,E2 -11304.497} C_VEL
LIN {X 0,Y 397.079,Z 401.022,A -85,B 0,C 180,E1 -11307.928,E2 -11307.928} C_VEL
LIN {X 0,Y 397.123,Z 401.019,A -85,B 0,C 180,E1 -11311.456,E2 -11311.456} C_VEL
LIN {X 0,Y 397.154,Z 401.013,A -85,B 0,C 180,E1 -11314.488,E2 -11314.488} C_VEL
LIN {X 0,Y 397.11,Z 401.022,A -85,B 0,C 180,E1 -11317.086,E2 -11317.086} C_VEL
LIN {X 0,Y 397.149,Z 401.013,A -85,B 0,C 180,E1 -11320.353,E2 -11320.353} C_VEL
LIN {X 0,Y 397.167,Z 401.012,A -85,B 0,C 180,E1 -11323.553,E2 -11323.553} C_VEL
LIN {X 0,Y 397.229,Z 401.005,A -85,B 0,C 180,E1 -11326.703,E2 -11326.703} C_VEL
LIN {X 0,Y 397.219,Z 401.004,A -85,B 0,C 180,E1 -11329.809,E2 -11329.809} C_VEL
LIN {X 0,Y 397.365,Z 400.99,A -85,B 0,C 180,E1 -11332.888,E2 -11332.888} C_VEL
LIN {X 0,Y 397.254,Z 401.004,A -85,B 0,C 180,E1 -11334.925,E2 -11334.925} C_VEL
LIN {X 0,Y 397.449,Z 400.975,A -85,B 0,C 180,E1 -11337.973,E2 -11337.973} C_VEL
LIN {X 0,Y 397.579,Z 400.96,A -85,B 0,C 180,E1 -11340,E2 -11340} C_VEL
LIN {X 0,Y 397.375,Z 400.988,A -85,B 0,C 180,E1 -11343.041,E2 -11343.041} C_VEL
LIN {X 0,Y 397.365,Z 400.99,A -85,B 0,C 180,E1 -11347.112,E2 -11347.112} C_VEL
LIN {X 0,Y 397.218,Z 401.005,A -85,B 0,C 180,E1 -11350.191,E2 -11350.191} C_VEL
LIN {X 0,Y 397.227,Z 401.005,A -85,B 0,C 180,E1 -11353.321,E2 -11353.321} C_VEL
LIN {X 0,Y 397.182,Z 401.012,A -85,B 0,C 180,E1 -11357.155,E2 -11357.155} C_VEL
LIN {X 0,Y 397.103,Z 401.023,A -85,B 0,C 180,E1 -11360.73,E2 -11360.73} C_VEL
LIN {X 0,Y 397.134,Z 401.015,A -85,B 0,C 180,E1 -11364.018,E2 -11364.018} C_VEL
LIN {X 0,Y 397.195,Z 401.008,A -85,B 0,C 180,E1 -11367.39,E2 -11367.39} C_VEL
LIN {X 0,Y 397.079,Z 401.026,A -85,B 0,C 180,E1 -11370.882,E2 -11370.882} C_VEL
LIN {X 0,Y 397.126,Z 401.019,A -85,B 0,C 180,E1 -11374.493,E2 -11374.493} C_VEL
LIN {X 0,Y 397.102,Z 401.021,A -85,B 0,C 180,E1 -11378.275,E2 -11378.275} C_VEL
LIN {X 0,Y 397.089,Z 401.023,A -85,B 0,C 180,E1 -11380.909,E2 -11380.909} C_VEL
LIN {X 0,Y 397.102,Z 401.018,A -85,B 0,C 180,E1 -11383.648,E2 -11383.648} C_VEL
LIN {X 0,Y 397.103,Z 401.023,A -85,B 0,C 180,E1 -11386.521,E2 -11386.521} C_VEL
LIN {X 0,Y 397.116,Z 401.021,A -85,B 0,C 180,E1 -11390.423,E2 -11390.423} C_VEL
LIN {X 0,Y 397.111,Z 401.021,A -85,B 0,C 180,E1 -11394.265,E2 -11394.265} C_VEL
LIN {X 0,Y 397.116,Z 401.021,A -85,B 0,C 180,E1 -11396.727,E2 -11396.727} C_VEL
LIN {X 0,Y 397.126,Z 401.019,A -85,B 0,C 180,E1 -11400.296,E2 -11400.296} C_VEL
LIN {X 0,Y 397.196,Z 401.011,A -85,B 0,C 180,E1 -11402.61,E2 -11402.61} C_VEL
LIN {X 0,Y 397.135,Z 401.017,A -85,B 0,C 180,E1 -11405.982,E2 -11405.982} C_VEL
LIN {X 0,Y 397.141,Z 401.015,A -85,B 0,C 180,E1 -11409.704,E2 -11409.704} C_VEL
LIN {X 0,Y 397.184,Z 401.01,A -85,B 0,C 180,E1 -11412.845,E2 -11412.845} C_VEL
LIN {X 0,Y 397.231,Z 401.005,A -85,B 0,C 180,E1 -11416.702,E2 -11416.702} C_VEL
LIN {X 0,Y 397.219,Z 401.005,A -85,B 0,C 180,E1 -11419.809,E2 -11419.809} C_VEL
LIN {X 0,Y 397.367,Z 400.987,A -85,B 0,C 180,E1 -11422.888,E2 -11422.888} C_VEL
LIN {X 0,Y 397.256,Z 401,A -85,B 0,C 180,E1 -11424.925,E2 -11424.925} C_VEL
LIN {X 0,Y 397.451,Z 400.978,A -85,B 0,C 180,E1 -11427.973,E2 -11427.973} C_VEL
LIN {X 0,Y 397.581,Z 400.963,A -85,B 0,C 180,E1 -11430,E2 -11430} C_VEL
LIN {X 0,Y 397.382,Z 400.984,A -85,B 0,C 180,E1 -11433.041,E2 -11433.041} C_VEL
LIN {X 0,Y 397.312,Z 400.996,A -85,B 0,C 180,E1 -11436.092,E2 -11436.092} C_VEL
LIN {X 0,Y 396.901,Z 401.047,A -85,B 0,C 180,E1 -11439.17,E2 -11439.17} C_VEL
LIN {X 0,Y 396.721,Z 404.365,A -85,B 0,C 180,E1 -11442.273,E2 -11442.273} C_VEL
LIN {X 0,Y 396.505,Z 408.062,A -85,B 0,C 180,E1 -11445.418,E2 -11445.418} C_VEL
LIN {X 0,Y 396.362,Z 410.603,A -85,B 0,C 180,E1 -11447.543,E2 -11447.543} C_VEL
LIN {X 0,Y 396.187,Z 414.546,A -85,B 0,C 180,E1 -11450.78,E2 -11450.78} C_VEL
LIN {X 0,Y 396.069,Z 418.632,A -85,B 0,C 180,E1 -11454.086,E2 -11454.086} C_VEL
LIN {X 0,Y 396.079,Z 419.139,A -85,B 0,C 180,E1 -11454.497,E2 -11454.497} C_VEL
LIN {X 0,Y 396.093,Z 420.439,A -85,B 0,C 180,E1 -11454.83,E2 -11454.83} C_VEL
LIN {X 0,Y 396.091,Z 423.426,A -85,B 0,C 180,E1 -11455.107,E2 -11455.107} C_VEL
LIN {X 0,Y 395.536,Z 437.759,A -85,B 0,C 180,E1 -11455.721,E2 -11455.721} C_VEL
LIN {X 0,Y 394.605,Z 445.721,A -85,B 0,C 180,E1 -11456.117,E2 -11456.117} C_VEL
LIN {X 0,Y 394.353,Z 448.303,A -85,B 0,C 180,E1 -11456.282,E2 -11456.282} C_VEL
LIN {X 0,Y 393.451,Z 461.138,A -85,B 0,C 180,E1 -11457.222,E2 -11457.222} C_VEL
LIN {X 0,Y 392.652,Z 472.587,A -85,B 0,C 180,E1 -11458.314,E2 -11458.314} C_VEL
LIN {X 0,Y 391.791,Z 482.971,A -85,B 0,C 180,E1 -11459.557,E2 -11459.557} C_VEL
LIN {X 0,Y 391.048,Z 492.078,A -85,B 0,C 180,E1 -11460.901,E2 -11460.901} C_VEL
LIN {X 0,Y 390.322,Z 500.4,A -85,B 0,C 180,E1 -11462.419,E2 -11462.419} C_VEL
LIN {X 0,Y 389.757,Z 507.277,A -85,B 0,C 180,E1 -11463.985,E2 -11463.985} C_VEL
LIN {X 0,Y 389.326,Z 513.164,A -85,B 0,C 180,E1 -11465.676,E2 -11465.676} C_VEL
LIN {X 0,Y 388.976,Z 517.625,A -85,B 0,C 180,E1 -11467.346,E2 -11467.346} C_VEL
LIN {X 0,Y 388.707,Z 521.229,A -85,B 0,C 180,E1 -11469.257,E2 -11469.257} C_VEL
LIN {X 0,Y 388.572,Z 522.938,A -85,B 0,C 180,E1 -11470.625,E2 -11470.625} C_VEL
LIN {X 0,Y 388.561,Z 523.966,A -85,B 0,C 180,E1 -11472.134,E2 -11472.134} C_VEL
LIN {X 0,Y 388.552,Z 524.158,A -85,B 0,C 180,E1 -11473.655,E2 -11473.655} C_VEL
LIN {X 0,Y 388.578,Z 523.528,A -85,B 0,C 180,E1 -11475.14,E2 -11475.14} C_VEL
LIN {X 0,Y 388.702,Z 522.116,A -85,B 0,C 180,E1 -11476.602,E2 -11476.602} C_VEL
LIN {X 0,Y 388.946,Z 519.902,A -85,B 0,C 180,E1 -11478.044,E2 -11478.044} C_VEL
LIN {X 0,Y 389.172,Z 516.913,A -85,B 0,C 180,E1 -11479.449,E2 -11479.449} C_VEL
LIN {X 0,Y 389.615,Z 511.949,A -85,B 0,C 180,E1 -11481.218,E2 -11481.218} C_VEL
LIN {X 0,Y 390.228,Z 505.288,A -85,B 0,C 180,E1 -11483.008,E2 -11483.008} C_VEL
LIN {X 0,Y 390.981,Z 497.342,A -85,B 0,C 180,E1 -11484.685,E2 -11484.685} C_VEL
LIN {X 0,Y 391.877,Z 488.119,A -85,B 0,C 180,E1 -11486.223,E2 -11486.223} C_VEL
LIN {X 0,Y 392.82,Z 478.304,A -85,B 0,C 180,E1 -11487.538,E2 -11487.538} C_VEL
LIN {X 0,Y 393.751,Z 467.773,A -85,B 0,C 180,E1 -11488.678,E2 -11488.678} C_VEL
LIN {X 0,Y 394.585,Z 456.513,A -85,B 0,C 180,E1 -11489.643,E2 -11489.643} C_VEL
LIN {X 0,Y 395.284,Z 447.003,A -85,B 0,C 180,E1 -11490.29,E2 -11490.29} C_VEL
LIN {X 0,Y 392.876,Z 435.006,A -85,B 0,C 180,E1 -11491.082,E2 -11491.082} C_VEL
LIN {X 0,Y 389.614,Z 422.987,A -85,B 0,C 180,E1 -11491.738,E2 -11491.738} C_VEL
LIN {X 0,Y 389.198,Z 421.097,A -85,B 0,C 180,E1 -11491.852,E2 -11491.852} C_VEL
LIN {X 0,Y 389.36,Z 416.944,A -85,B 0,C 180,E1 -11495.471,E2 -11495.471} C_VEL
LIN {X 0,Y 389.553,Z 413.181,A -85,B 0,C 180,E1 -11498.849,E2 -11498.849} C_VEL
LIN {X 0,Y 389.795,Z 409.596,A -85,B 0,C 180,E1 -11502.151,E2 -11502.151} C_VEL
LIN {X 0,Y 390.036,Z 406.195,A -85,B 0,C 180,E1 -11505.389,E2 -11505.389} C_VEL
LIN {X 0,Y 390.181,Z 404.03,A -85,B 0,C 180,E1 -11507.517,E2 -11507.517} C_VEL
LIN {X 0,Y 390.121,Z 401.981,A -85,B 0,C 180,E1 -11509.622,E2 -11509.622} C_VEL
LIN {X 0,Y 390.314,Z 401.869,A -85,B 0,C 180,E1 -11512.759,E2 -11512.759} C_VEL
LIN {X 0,Y 390.224,Z 401.879,A -85,B 0,C 180,E1 -11514.834,E2 -11514.834} C_VEL
LIN {X 0,Y 390.417,Z 401.857,A -85,B 0,C 180,E1 -11517.937,E2 -11517.937} C_VEL
LIN {X 0,Y 390.548,Z 401.839,A -85,B 0,C 180,E1 -11520,E2 -11520} C_VEL
LIN {X 0,Y 390.311,Z 401.869,A -85,B 0,C 180,E1 -11523.097,E2 -11523.097} C_VEL
LIN {X 0,Y 390.326,Z 401.867,A -85,B 0,C 180,E1 -11526.202,E2 -11526.202} C_VEL
LIN {X 0,Y 390.31,Z 401.868,A -85,B 0,C 180,E1 -11528.282,E2 -11528.282} C_VEL
LIN {X 0,Y 390.167,Z 401.886,A -85,B 0,C 180,E1 -11532.483,E2 -11532.483} C_VEL
LIN {X 0,Y 390.135,Z 401.889,A -85,B 0,C 180,E1 -11535.677,E2 -11535.677} C_VEL
LIN {X 0,Y 390.102,Z 401.894,A -85,B 0,C 180,E1 -11538.922,E2 -11538.922} C_VEL
LIN {X 0,Y 390.036,Z 401.902,A -85,B 0,C 180,E1 -11542.234,E2 -11542.234} C_VEL
LIN {X 0,Y 390.116,Z 401.893,A -85,B 0,C 180,E1 -11545.744,E2 -11545.744} C_VEL
LIN {X 0,Y 390.062,Z 401.899,A -85,B 0,C 180,E1 -11549.109,E2 -11549.109} C_VEL
LIN {X 0,Y 390.041,Z 401.902,A -85,B 0,C 180,E1 -11552.722,E2 -11552.722} C_VEL
LIN {X 0,Y 390.055,Z 401.902,A -85,B 0,C 180,E1 -11555.826,E2 -11555.826} C_VEL
LIN {X 0,Y 390.072,Z 401.901,A -85,B 0,C 180,E1 -11559.22,E2 -11559.22} C_VEL
LIN {X 0,Y 390.078,Z 401.899,A -85,B 0,C 180,E1 -11562.381,E2 -11562.381} C_VEL
LIN {X 0,Y 390.052,Z 401.915,A -85,B 0,C 180,E1 -11566.115,E2 -11566.115} C_VEL
LIN {X 0,Y 390.922,Z 406.744,A -85,B 0,C 180,E1 -11569.669,E2 -11569.669} C_VEL
LIN {X 0,Y 391.544,Z 410.815,A -85,B 0,C 180,E1 -11572.391,E2 -11572.391} C_VEL
LIN {X 0,Y 391.717,Z 415.005,A -85,B 0,C 180,E1 -11574.962,E2 -11574.962} C_VEL
LIN {X 0,Y 391.034,Z 421.435,A -85,B 0,C 180,E1 -11578.587,E2 -11578.587} C_VEL
LIN {X 0,Y 390.416,Z 428,A -85,B 0,C 180,E1 -11582.094,E2 -11582.094} C_VEL
LIN {X 0,Y 389.955,Z 434.676,A -85,B 0,C 180,E1 -11585.512,E2 -11585.512} C_VEL
LIN {X 0,Y 389.54,Z 441.449,A -85,B 0,C 180,E1 -11588.849,E2 -11588.849} C_VEL
LIN {X 0,Y 389.285,Z 446.264,A -85,B 0,C 180,E1 -11591.173,E2 -11591.173} C_VEL
LIN {X 0,Y 392.146,Z 460.469,A -85,B 0,C 180,E1 -11591.826,E2 -11591.826} C_VEL
LIN {X 0,Y 393.681,Z 472.866,A -85,B 0,C 180,E1 -11592.549,E2 -11592.549} C_VEL
LIN {X 0,Y 394.251,Z 480.263,A -85,B 0,C 180,E1 -11593.061,E2 -11593.061} C_VEL
LIN {X 0,Y 393.341,Z 491.47,A -85,B 0,C 180,E1 -11593.923,E2 -11593.923} C_VEL
LIN {X 0,Y 392.295,Z 503.211,A -85,B 0,C 180,E1 -11595.077,E2 -11595.077} C_VEL
LIN {X 0,Y 391.485,Z 513.21,A -85,B 0,C 180,E1 -11596.305,E2 -11596.305} C_VEL
LIN {X 0,Y 390.734,Z 521.456,A -85,B 0,C 180,E1 -11597.536,E2 -11597.536} C_VEL
LIN {X 0,Y 389.883,Z 529.963,A -85,B 0,C 180,E1 -11599.09,E2 -11599.09} C_VEL
LIN {X 0,Y 389.376,Z 536.837,A -85,B 0,C 180,E1 -11600.652,E2 -11600.652} C_VEL
LIN {X 0,Y 389.022,Z 542.35,A -85,B 0,C 180,E1 -11602.213,E2 -11602.213} C_VEL
LIN {X 0,Y 388.797,Z 546.8,A -85,B 0,C 180,E1 -11603.826,E2 -11603.826} C_VEL
LIN {X 0,Y 388.745,Z 548.974,A -85,B 0,C 180,E1 -11604.814,E2 -11604.814} C_VEL
LIN {X 0,Y 388.704,Z 550.8,A -85,B 0,C 180,E1 -11605.853,E2 -11605.853} C_VEL
LIN {X 0,Y 388.703,Z 553.178,A -85,B 0,C 180,E1 -11607.928,E2 -11607.928} C_VEL
LIN {X 0,Y 388.74,Z 553.775,A -85,B 0,C 180,E1 -11608.964,E2 -11608.964} C_VEL
LIN {X 0,Y 388.726,Z 553.933,A -85,B 0,C 180,E1 -11610,E2 -11610} C_VEL
LIN {X 0,Y 388.74,Z 553.684,A -85,B 0,C 180,E1 -11611.036,E2 -11611.036} C_VEL
LIN {X 0,Y 388.721,Z 553.042,A -85,B 0,C 180,E1 -11612.073,E2 -11612.073} C_VEL
LIN {X 0,Y 388.653,Z 552.002,A -85,B 0,C 180,E1 -11613.11,E2 -11613.11} C_VEL
LIN {X 0,Y 388.707,Z 550.51,A -85,B 0,C 180,E1 -11614.148,E2 -11614.148} C_VEL
LIN {X 0,Y 388.732,Z 547.335,A -85,B 0,C 180,E1 -11615.76,E2 -11615.76} C_VEL
LIN {X 0,Y 388.935,Z 543.348,A -85,B 0,C 180,E1 -11617.267,E2 -11617.267} C_VEL
LIN {X 0,Y 389.285,Z 537.029,A -85,B 0,C 180,E1 -11619.089,E2 -11619.089} C_VEL
LIN {X 0,Y 389.773,Z 530.145,A -85,B 0,C 180,E1 -11620.651,E2 -11620.651} C_VEL
LIN {X 0,Y 390.358,Z 523.12,A -85,B 0,C 180,E1 -11621.95,E2 -11621.95} C_VEL
LIN {X 0,Y 391.046,Z 514.663,A -85,B 0,C 180,E1 -11623.247,E2 -11623.247} C_VEL
LIN {X 0,Y 391.864,Z 504.226,A -85,B 0,C 180,E1 -11624.542,E2 -11624.542} C_VEL
LIN {X 0,Y 392.802,Z 492.517,A -85,B 0,C 180,E1 -11625.701,E2 -11625.701} C_VEL
LIN {X 0,Y 393.673,Z 480.871,A -85,B 0,C 180,E1 -11626.597,E2 -11626.597} C_VEL
LIN {X 0,Y 393.248,Z 473.724,A -85,B 0,C 180,E1 -11627.074,E2 -11627.074} C_VEL
LIN {X 0,Y 391.533,Z 460.419,A -85,B 0,C 180,E1 -11627.817,E2 -11627.817} C_VEL
LIN {X 0,Y 389.249,Z 447.29,A -85,B 0,C 180,E1 -11628.355,E2 -11628.355} C_VEL
LIN {X 0,Y 389.608,Z 440.304,A -85,B 0,C 180,E1 -11631.703,E2 -11631.703} C_VEL
LIN {X 0,Y 389.989,Z 433.449,A -85,B 0,C 180,E1 -11635.056,E2 -11635.056} C_VEL
LIN {X 0,Y 390.42,Z 427.346,A -85,B 0,C 180,E1 -11638.108,E2 -11638.108} C_VEL
LIN {X 0,Y 390.969,Z 420.888,A -85,B 0,C 180,E1 -11641.42,E2 -11641.42} C_VEL
LIN {X 0,Y 391.465,Z 415.384,A -85,B 0,C 180,E1 -11644.326,E2 -11644.326} C_VEL
LIN {X 0,Y 391.467,Z 410.599,A -85,B 0,C 180,E1 -11646.972,E2 -11646.972} C_VEL
LIN {X 0,Y 390.94,Z 406.498,A -85,B 0,C 180,E1 -11649.374,E2 -11649.374} C_VEL
LIN {X 0,Y 390.064,Z 401.9,A -85,B 0,C 180,E1 -11652.294,E2 -11652.294} C_VEL
LIN {X 0,Y 390.046,Z 401.902,A -85,B 0,C 180,E1 -11655.354,E2 -11655.354} C_VEL
LIN {X 0,Y 390.032,Z 401.899,A -85,B 0,C 180,E1 -11658.187,E2 -11658.187} C_VEL
LIN {X 0,Y 390.09,Z 401.895,A -85,B 0,C 180,E1 -11660.907,E2 -11660.907} C_VEL
LIN {X 0,Y 390.086,Z 401.895,A -85,B 0,C 180,E1 -11664.793,E2 -11664.793} C_VEL
LIN {X 0,Y 390.024,Z 401.901,A -85,B 0,C 180,E1 -11668.496,E2 -11668.496} C_VEL
LIN {X 0,Y 390.118,Z 401.888,A -85,B 0,C 180,E1 -11672.07,E2 -11672.07} C_VEL
LIN {X 0,Y 390.081,Z 401.896,A -85,B 0,C 180,E1 -11675.519,E2 -11675.519} C_VEL
LIN {X 0,Y 390.056,Z 401.9,A -85,B 0,C 180,E1 -11678.878,E2 -11678.878} C_VEL
LIN {X 0,Y 390.129,Z 401.887,A -85,B 0,C 180,E1 -11682.167,E2 -11682.167} C_VEL
LIN {X 0,Y 390.145,Z 401.888,A -85,B 0,C 180,E1 -11685.393,E2 -11685.393} C_VEL
LIN {X 0,Y 390.149,Z 401.887,A -85,B 0,C 180,E1 -11688.571,E2 -11688.571} C_VEL
LIN {X 0,Y 390.345,Z 401.86,A -85,B 0,C 180,E1 -11691.993,E2 -11691.993} C_VEL
LIN {X 0,Y 390.226,Z 401.879,A -85,B 0,C 180,E1 -11694.833,E2 -11694.833} C_VEL
LIN {X 0,Y 390.418,Z 401.851,A -85,B 0,C 180,E1 -11697.937,E2 -11697.937} C_VEL
LIN {X 0,Y 390.549,Z 401.835,A -85,B 0,C 180,E1 -11700,E2 -11700} C_VEL
LIN {X 0,Y 390.31,Z 401.869,A -85,B 0,C 180,E1 -11703.096,E2 -11703.096} C_VEL
LIN {X 0,Y 390.31,Z 401.864,A -85,B 0,C 180,E1 -11706.635,E2 -11706.635} C_VEL
LIN {X 0,Y 390.206,Z 401.88,A -85,B 0,C 180,E1 -11709.329,E2 -11709.329} C_VEL
LIN {X 0,Y 390.195,Z 401.88,A -85,B 0,C 180,E1 -11713.438,E2 -11713.438} C_VEL
LIN {X 0,Y 390.149,Z 401.887,A -85,B 0,C 180,E1 -11717.308,E2 -11717.308} C_VEL
LIN {X 0,Y 390.088,Z 401.895,A -85,B 0,C 180,E1 -11720.47,E2 -11720.47} C_VEL
LIN {X 0,Y 390.09,Z 401.893,A -85,B 0,C 180,E1 -11723.351,E2 -11723.351} C_VEL
LIN {X 0,Y 390.114,Z 401.893,A -85,B 0,C 180,E1 -11726.768,E2 -11726.768} C_VEL
LIN {X 0,Y 390.04,Z 401.901,A -85,B 0,C 180,E1 -11730.3,E2 -11730.3} C_VEL
LIN {X 0,Y 390.069,Z 401.895,A -85,B 0,C 180,E1 -11734.025,E2 -11734.025} C_VEL
LIN {X 0,Y 390.043,Z 401.897,A -85,B 0,C 180,E1 -11737.551,E2 -11737.551} C_VEL
LIN {X 0,Y 390.057,Z 401.9,A -85,B 0,C 180,E1 -11740.821,E2 -11740.821} C_VEL
LIN {X 0,Y 390.055,Z 401.896,A -85,B 0,C 180,E1 -11743.886,E2 -11743.886} C_VEL
LIN {X 0,Y 390.058,Z 401.9,A -85,B 0,C 180,E1 -11746.79,E2 -11746.79} C_VEL
LIN {X 0,Y 390.057,Z 401.895,A -85,B 0,C 180,E1 -11749.561,E2 -11749.561} C_VEL
LIN {X 0,Y 390.047,Z 401.901,A -85,B 0,C 180,E1 -11752.449,E2 -11752.449} C_VEL
LIN {X 0,Y 390.07,Z 401.895,A -85,B 0,C 180,E1 -11755.975,E2 -11755.975} C_VEL
LIN {X 0,Y 390.048,Z 401.898,A -85,B 0,C 180,E1 -11759.869,E2 -11759.869} C_VEL
LIN {X 0,Y 390.115,Z 401.889,A -85,B 0,C 180,E1 -11763.232,E2 -11763.232} C_VEL
LIN {X 0,Y 390.108,Z 401.893,A -85,B 0,C 180,E1 -11766.75,E2 -11766.75} C_VEL
LIN {X 0,Y 390.106,Z 401.892,A -85,B 0,C 180,E1 -11769.983,E2 -11769.983} C_VEL
LIN {X 0,Y 390.14,Z 401.885,A -85,B 0,C 180,E1 -11773.248,E2 -11773.248} C_VEL
LIN {X 0,Y 390.196,Z 401.882,A -85,B 0,C 180,E1 -11776.561,E2 -11776.561} C_VEL
LIN {X 0,Y 390.207,Z 401.881,A -85,B 0,C 180,E1 -11780.671,E2 -11780.671} C_VEL
LIN {X 0,Y 390.321,Z 401.866,A -85,B 0,C 180,E1 -11782.759,E2 -11782.759} C_VEL
LIN {X 0,Y 390.228,Z 401.876,A -85,B 0,C 180,E1 -11784.833,E2 -11784.833} C_VEL
LIN {X 0,Y 390.419,Z 401.854,A -85,B 0,C 180,E1 -11787.936,E2 -11787.936} C_VEL
LIN {X 0,Y 390.55,Z 401.838,A -85,B 0,C 180,E1 -11790,E2 -11790} C_VEL
LIN {X 0,Y 390.316,Z 401.864,A -85,B 0,C 180,E1 -11793.096,E2 -11793.096} C_VEL
LIN {X 0,Y 390.258,Z 401.875,A -85,B 0,C 180,E1 -11796.203,E2 -11796.203} C_VEL
LIN {X 0,Y 389.812,Z 401.93,A -85,B 0,C 180,E1 -11799.338,E2 -11799.338} C_VEL
LIN {X 0,Y 389.643,Z 406.12,A -85,B 0,C 180,E1 -11803.094,E2 -11803.094} C_VEL
LIN {X 0,Y 389.38,Z 410.631,A -85,B 0,C 180,E1 -11806.94,E2 -11806.94} C_VEL
LIN {X 0,Y 389.175,Z 414.392,A -85,B 0,C 180,E1 -11810.107,E2 -11810.107} C_VEL
LIN {X 0,Y 389.023,Z 418.449,A -85,B 0,C 180,E1 -11813.418,E2 -11813.418} C_VEL
LIN {X 0,Y 389.027,Z 420.133,A -85,B 0,C 180,E1 -11814.741,E2 -11814.741} C_VEL
LIN {X 0,Y 392.041,Z 433.29,A -85,B 0,C 180,E1 -11815.357,E2 -11815.357} C_VEL
LIN {X 0,Y 394.185,Z 443.997,A -85,B 0,C 180,E1 -11816.007,E2 -11816.007} C_VEL
LIN {X 0,Y 394.353,Z 448.303,A -85,B 0,C 180,E1 -11816.282,E2 -11816.282} C_VEL
LIN {X 0,Y 393.436,Z 451.956,A -85,B 0,C 180,E1 -11816.492,E2 -11816.492} C_VEL
LIN {X 0,Y 387.086,Z 463.096,A -85,B 0,C 180,E1 -11817.136,E2 -11817.136} C_VEL
LIN {X 0,Y 386.223,Z 466.406,A -85,B 0,C 180,E1 -11817.417,E2 -11817.417} C_VEL
LIN {X 0,Y 385.398,Z 477.236,A -85,B 0,C 180,E1 -11818.575,E2 -11818.575} C_VEL
LIN {X 0,Y 384.566,Z 486.956,A -85,B 0,C 180,E1 -11819.867,E2 -11819.867} C_VEL
LIN {X 0,Y 383.847,Z 494.877,A -85,B 0,C 180,E1 -11821.147,E2 -11821.147} C_VEL
LIN {X 0,Y 383.221,Z 501.715,A -85,B 0,C 180,E1 -11822.477,E2 -11822.477} C_VEL
LIN {X 0,Y 382.611,Z 509.088,A -85,B 0,C 180,E1 -11824.251,E2 -11824.251} C_VEL
LIN {X 0,Y 382.155,Z 514.818,A -85,B 0,C 180,E1 -11826.049,E2 -11826.049} C_VEL
LIN {X 0,Y 381.845,Z 518.77,A -85,B 0,C 180,E1 -11827.68,E2 -11827.68} C_VEL
LIN {X 0,Y 381.605,Z 521.662,A -85,B 0,C 180,E1 -11829.33,E2 -11829.33} C_VEL
LIN {X 0,Y 381.476,Z 523.493,A -85,B 0,C 180,E1 -11830.944,E2 -11830.944} C_VEL
LIN {X 0,Y 381.452,Z 524.453,A -85,B 0,C 180,E1 -11832.976,E2 -11832.976} C_VEL
LIN {X 0,Y 381.457,Z 524.226,A -85,B 0,C 180,E1 -11834.435,E2 -11834.435} C_VEL
LIN {X 0,Y 381.529,Z 523.229,A -85,B 0,C 180,E1 -11835.922,E2 -11835.922} C_VEL
LIN {X 0,Y 381.727,Z 521.4,A -85,B 0,C 180,E1 -11837.428,E2 -11837.428} C_VEL
LIN {X 0,Y 382.11,Z 517.528,A -85,B 0,C 180,E1 -11839.453,E2 -11839.453} C_VEL
LIN {X 0,Y 382.594,Z 512.386,A -85,B 0,C 180,E1 -11841.35,E2 -11841.35} C_VEL
LIN {X 0,Y 383.194,Z 506.428,A -85,B 0,C 180,E1 -11843.016,E2 -11843.016} C_VEL
LIN {X 0,Y 383.831,Z 500.03,A -85,B 0,C 180,E1 -11844.454,E2 -11844.454} C_VEL
LIN {X 0,Y 384.671,Z 491.673,A -85,B 0,C 180,E1 -11845.977,E2 -11845.977} C_VEL
LIN {X 0,Y 385.568,Z 483.084,A -85,B 0,C 180,E1 -11847.253,E2 -11847.253} C_VEL
LIN {X 0,Y 386.544,Z 473.124,A -85,B 0,C 180,E1 -11848.464,E2 -11848.464} C_VEL
LIN {X 0,Y 387.4,Z 462.872,A -85,B 0,C 180,E1 -11849.472,E2 -11849.472} C_VEL
LIN {X 0,Y 388.196,Z 451.737,A -85,B 0,C 180,E1 -11850.342,E2 -11850.342} C_VEL
LIN {X 0,Y 388.402,Z 447.034,A -85,B 0,C 180,E1 -11850.656,E2 -11850.656} C_VEL
LIN {X 0,Y 385.759,Z 434.606,A -85,B 0,C 180,E1 -11851.504,E2 -11851.504} C_VEL
LIN {X 0,Y 382.166,Z 421.41,A -85,B 0,C 180,E1 -11852.25,E2 -11852.25} C_VEL
LIN {X 0,Y 382.349,Z 417.036,A -85,B 0,C 180,E1 -11856.147,E2 -11856.147} C_VEL
LIN {X 0,Y 382.572,Z 413.288,A -85,B 0,C 180,E1 -11859.572,E2 -11859.572} C_VEL
LIN {X 0,Y 382.842,Z 409.757,A -85,B 0,C 180,E1 -11862.919,E2 -11862.919} C_VEL
LIN {X 0,Y 383.1,Z 406.127,A -85,B 0,C 180,E1 -11866.477,E2 -11866.477} C_VEL
LIN {X 0,Y 383.12,Z 403.273,A -85,B 0,C 180,E1 -11869.43,E2 -11869.43} C_VEL
LIN {X 0,Y 383.131,Z 402.768,A -85,B 0,C 180,E1 -11870.497,E2 -11870.497} C_VEL
LIN {X 0,Y 383.27,Z 402.747,A -85,B 0,C 180,E1 -11872.625,E2 -11872.625} C_VEL
LIN {X 0,Y 383.196,Z 402.755,A -85,B 0,C 180,E1 -11874.739,E2 -11874.739} C_VEL
LIN {X 0,Y 383.384,Z 402.733,A -85,B 0,C 180,E1 -11877.899,E2 -11877.899} C_VEL
LIN {X 0,Y 383.517,Z 402.715,A -85,B 0,C 180,E1 -11880,E2 -11880} C_VEL
LIN {X 0,Y 383.248,Z 402.748,A -85,B 0,C 180,E1 -11883.154,E2 -11883.154} C_VEL
LIN {X 0,Y 383.283,Z 402.744,A -85,B 0,C 180,E1 -11886.316,E2 -11886.316} C_VEL
LIN {X 0,Y 383.256,Z 402.747,A -85,B 0,C 180,E1 -11888.436,E2 -11888.436} C_VEL
LIN {X 0,Y 383.093,Z 402.767,A -85,B 0,C 180,E1 -11891.642,E2 -11891.642} C_VEL
LIN {X 0,Y 383.106,Z 402.765,A -85,B 0,C 180,E1 -11894.882,E2 -11894.882} C_VEL
LIN {X 0,Y 383.085,Z 402.769,A -85,B 0,C 180,E1 -11898.173,E2 -11898.173} C_VEL
LIN {X 0,Y 382.989,Z 402.78,A -85,B 0,C 180,E1 -11901.531,E2 -11901.531} C_VEL
LIN {X 0,Y 383.049,Z 402.773,A -85,B 0,C 180,E1 -11904.961,E2 -11904.961} C_VEL
LIN {X 0,Y 383.046,Z 402.773,A -85,B 0,C 180,E1 -11908.492,E2 -11908.492} C_VEL
LIN {X 0,Y 383.008,Z 402.779,A -85,B 0,C 180,E1 -11912.15,E2 -11912.15} C_VEL
LIN {X 0,Y 383.015,Z 402.778,A -85,B 0,C 180,E1 -11914.668,E2 -11914.668} C_VEL
LIN {X 0,Y 383.001,Z 402.782,A -85,B 0,C 180,E1 -11917.905,E2 -11917.905} C_VEL
LIN {X 0,Y 383.012,Z 402.78,A -85,B 0,C 180,E1 -11921.344,E2 -11921.344} C_VEL
LIN {X 0,Y 382.994,Z 402.78,A -85,B 0,C 180,E1 -11924.304,E2 -11924.304} C_VEL
LIN {X 0,Y 383.016,Z 402.974,A -85,B 0,C 180,E1 -11925.793,E2 -11925.793} C_VEL
LIN {X 0,Y 383.718,Z 406.822,A -85,B 0,C 180,E1 -11928.75,E2 -11928.75} C_VEL
LIN {X 0,Y 384.452,Z 411.225,A -85,B 0,C 180,E1 -11931.82,E2 -11931.82} C_VEL
LIN {X 0,Y 384.71,Z 414.979,A -85,B 0,C 180,E1 -11934.227,E2 -11934.227} C_VEL
LIN {X 0,Y 384.491,Z 418.147,A -85,B 0,C 180,E1 -11936.118,E2 -11936.118} C_VEL
LIN {X 0,Y 383.861,Z 423.912,A -85,B 0,C 180,E1 -11939.374,E2 -11939.374} C_VEL
LIN {X 0,Y 383.198,Z 431.2,A -85,B 0,C 180,E1 -11943.299,E2 -11943.299} C_VEL
LIN {X 0,Y 382.763,Z 437.683,A -85,B 0,C 180,E1 -11946.645,E2 -11946.645} C_VEL
LIN {X 0,Y 382.31,Z 444.704,A -85,B 0,C 180,E1 -11950.143,E2 -11950.143} C_VEL
LIN {X 0,Y 382.242,Z 446.13,A -85,B 0,C 180,E1 -11950.776,E2 -11950.776} C_VEL
LIN {X 0,Y 385.103,Z 459.775,A -85,B 0,C 180,E1 -11951.423,E2 -11951.423} C_VEL
LIN {X 0,Y 386.658,Z 471.364,A -85,B 0,C 180,E1 -11952.113,E2 -11952.113} C_VEL
LIN {X 0,Y 387.399,Z 480.49,A -85,B 0,C 180,E1 -11952.756,E2 -11952.756} C_VEL
LIN {X 0,Y 386.534,Z 491.511,A -85,B 0,C 180,E1 -11953.632,E2 -11953.632} C_VEL
LIN {X 0,Y 385.401,Z 503.193,A -85,B 0,C 180,E1 -11954.804,E2 -11954.804} C_VEL
LIN {X 0,Y 384.531,Z 513.32,A -85,B 0,C 180,E1 -11956.076,E2 -11956.076} C_VEL
LIN {X 0,Y 383.632,Z 522.874,A -85,B 0,C 180,E1 -11957.57,E2 -11957.57} C_VEL
LIN {X 0,Y 382.791,Z 531.067,A -85,B 0,C 180,E1 -11959.153,E2 -11959.153} C_VEL
LIN {X 0,Y 382.359,Z 536.661,A -85,B 0,C 180,E1 -11960.479,E2 -11960.479} C_VEL
LIN {X 0,Y 381.948,Z 542.148,A -85,B 0,C 180,E1 -11962.068,E2 -11962.068} C_VEL
LIN {X 0,Y 381.69,Z 546.978,A -85,B 0,C 180,E1 -11963.878,E2 -11963.878} C_VEL
LIN {X 0,Y 381.629,Z 550.556,A -85,B 0,C 180,E1 -11965.776,E2 -11965.776} C_VEL
LIN {X 0,Y 381.601,Z 552.922,A -85,B 0,C 180,E1 -11967.889,E2 -11967.889} C_VEL
LIN {X 0,Y 381.67,Z 553.511,A -85,B 0,C 180,E1 -11968.945,E2 -11968.945} C_VEL
LIN {X 0,Y 381.656,Z 553.657,A -85,B 0,C 180,E1 -11970,E2 -11970} C_VEL
LIN {X 0,Y 381.672,Z 553.4,A -85,B 0,C 180,E1 -11971.055,E2 -11971.055} C_VEL
LIN {X 0,Y 381.62,Z 552.749,A -85,B 0,C 180,E1 -11972.111,E2 -11972.111} C_VEL
LIN {X 0,Y 381.563,Z 551.699,A -85,B 0,C 180,E1 -11973.168,E2 -11973.168} C_VEL
LIN {X 0,Y 381.633,Z 550.193,A -85,B 0,C 180,E1 -11974.225,E2 -11974.225} C_VEL
LIN {X 0,Y 381.69,Z 546.398,A -85,B 0,C 180,E1 -11976.121,E2 -11976.121} C_VEL
LIN {X 0,Y 381.943,Z 541.362,A -85,B 0,C 180,E1 -11977.933,E2 -11977.933} C_VEL
LIN {X 0,Y 382.398,Z 534.507,A -85,B 0,C 180,E1 -11979.788,E2 -11979.788} C_VEL
LIN {X 0,Y 382.935,Z 527.05,A -85,B 0,C 180,E1 -11981.379,E2 -11981.379} C_VEL
LIN {X 0,Y 383.692,Z 519.464,A -85,B 0,C 180,E1 -11982.698,E2 -11982.698} C_VEL
LIN {X 0,Y 384.517,Z 509.949,A -85,B 0,C 180,E1 -11984.059,E2 -11984.059} C_VEL
LIN {X 0,Y 385.267,Z 500.082,A -85,B 0,C 180,E1 -11985.203,E2 -11985.203} C_VEL
LIN {X 0,Y 386.186,Z 488.827,A -85,B 0,C 180,E1 -11986.249,E2 -11986.249} C_VEL
LIN {X 0,Y 386.794,Z 478.945,A -85,B 0,C 180,E1 -11986.985,E2 -11986.985} C_VEL
LIN {X 0,Y 385.303,Z 465.964,A -85,B 0,C 180,E1 -11987.82,E2 -11987.82} C_VEL
LIN {X 0,Y 383.254,Z 453.251,A -85,B 0,C 180,E1 -11988.435,E2 -11988.435} C_VEL
LIN {X 0,Y 382.183,Z 446.999,A -85,B 0,C 180,E1 -11988.686,E2 -11988.686} C_VEL
LIN {X 0,Y 382.583,Z 440.004,A -85,B 0,C 180,E1 -11992.122,E2 -11992.122} C_VEL
LIN {X 0,Y 383.036,Z 432.336,A -85,B 0,C 180,E1 -11995.965,E2 -11995.965} C_VEL
LIN {X 0,Y 383.639,Z 425.187,A -85,B 0,C 180,E1 -11999.645,E2 -11999.645} C_VEL
LIN {X 0,Y 384.27,Z 418.347,A -85,B 0,C 180,E1 -12003.276,E2 -12003.276} C_VEL
LIN {X 0,Y 384.527,Z 413.782,A -85,B 0,C 180,E1 -12005.794,E2 -12005.794} C_VEL
LIN {X 0,Y 384.224,Z 409.733,A -85,B 0,C 180,E1 -12008.137,E2 -12008.137} C_VEL
LIN {X 0,Y 383.342,Z 404.578,A -85,B 0,C 180,E1 -12011.301,E2 -12011.301} C_VEL
LIN {X 0,Y 383.039,Z 402.774,A -85,B 0,C 180,E1 -12012.577,E2 -12012.577} C_VEL
LIN {X 0,Y 382.999,Z 402.78,A -85,B 0,C 180,E1 -12015.789,E2 -12015.789} C_VEL
LIN {X 0,Y 382.989,Z 402.779,A -85,B 0,C 180,E1 -12018.796,E2 -12018.796} C_VEL
LIN {X 0,Y 383,Z 402.775,A -85,B 0,C 180,E1 -12022.096,E2 -12022.096} C_VEL
LIN {X 0,Y 383.019,Z 402.777,A -85,B 0,C 180,E1 -12025.332,E2 -12025.332} C_VEL
LIN {X 0,Y 382.984,Z 402.782,A -85,B 0,C 180,E1 -12029.081,E2 -12029.081} C_VEL
LIN {X 0,Y 383.058,Z 402.77,A -85,B 0,C 180,E1 -12032.698,E2 -12032.698} C_VEL
LIN {X 0,Y 383.053,Z 402.773,A -85,B 0,C 180,E1 -12035.04,E2 -12035.04} C_VEL
LIN {X 0,Y 382.994,Z 402.776,A -85,B 0,C 180,E1 -12038.469,E2 -12038.469} C_VEL
LIN {X 0,Y 383.064,Z 402.768,A -85,B 0,C 180,E1 -12041.826,E2 -12041.826} C_VEL
LIN {X 0,Y 383.111,Z 402.765,A -85,B 0,C 180,E1 -12045.118,E2 -12045.118} C_VEL
LIN {X 0,Y 383.098,Z 402.764,A -85,B 0,C 180,E1 -12048.358,E2 -12048.358} C_VEL
LIN {X 0,Y 383.305,Z 402.737,A -85,B 0,C 180,E1 -12051.933,E2 -12051.933} C_VEL
LIN {X 0,Y 383.199,Z 402.754,A -85,B 0,C 180,E1 -12054.738,E2 -12054.738} C_VEL
LIN {X 0,Y 383.386,Z 402.727,A -85,B 0,C 180,E1 -12057.899,E2 -12057.899} C_VEL
LIN {X 0,Y 383.518,Z 402.711,A -85,B 0,C 180,E1 -12060,E2 -12060} C_VEL
LIN {X 0,Y 383.247,Z 402.748,A -85,B 0,C 180,E1 -12063.154,E2 -12063.154} C_VEL
LIN {X 0,Y 383.27,Z 402.741,A -85,B 0,C 180,E1 -12066.629,E2 -12066.629} C_VEL
LIN {X 0,Y 383.261,Z 402.744,A -85,B 0,C 180,E1 -12068.436,E2 -12068.436} C_VEL
LIN {X 0,Y 383.098,Z 402.763,A -85,B 0,C 180,E1 -12071.642,E2 -12071.642} C_VEL
LIN {X 0,Y 383.111,Z 402.765,A -85,B 0,C 180,E1 -12074.882,E2 -12074.882} C_VEL
LIN {X 0,Y 383.09,Z 402.765,A -85,B 0,C 180,E1 -12078.172,E2 -12078.172} C_VEL
LIN {X 0,Y 382.994,Z 402.776,A -85,B 0,C 180,E1 -12081.531,E2 -12081.531} C_VEL
LIN {X 0,Y 383.053,Z 402.772,A -85,B 0,C 180,E1 -12084.96,E2 -12084.96} C_VEL
LIN {X 0,Y 383.041,Z 402.773,A -85,B 0,C 180,E1 -12088.493,E2 -12088.493} C_VEL
LIN {X 0,Y 383.01,Z 402.775,A -85,B 0,C 180,E1 -12092.15,E2 -12092.15} C_VEL
LIN {X 0,Y 383.019,Z 402.778,A -85,B 0,C 180,E1 -12094.668,E2 -12094.668} C_VEL
LIN {X 0,Y 382.999,Z 402.775,A -85,B 0,C 180,E1 -12097.904,E2 -12097.904} C_VEL
LIN {X 0,Y 382.984,Z 402.778,A -85,B 0,C 180,E1 -12101.347,E2 -12101.347} C_VEL
LIN {X 0,Y 382.997,Z 402.778,A -85,B 0,C 180,E1 -12104.303,E2 -12104.303} C_VEL
LIN {X 0,Y 383.011,Z 402.775,A -85,B 0,C 180,E1 -12107.24,E2 -12107.24} C_VEL
LIN {X 0,Y 383.017,Z 402.777,A -85,B 0,C 180,E1 -12110.413,E2 -12110.413} C_VEL
LIN {X 0,Y 383.028,Z 402.773,A -85,B 0,C 180,E1 -12114.045,E2 -12114.045} C_VEL
LIN {X 0,Y 382.988,Z 402.777,A -85,B 0,C 180,E1 -12117.578,E2 -12117.578} C_VEL
LIN {X 0,Y 382.994,Z 402.78,A -85,B 0,C 180,E1 -12120.3,E2 -12120.3} C_VEL
LIN {X 0,Y 383.082,Z 402.767,A -85,B 0,C 180,E1 -12124.021,E2 -12124.021} C_VEL
LIN {X 0,Y 383.01,Z 402.773,A -85,B 0,C 180,E1 -12127.335,E2 -12127.335} C_VEL
LIN {X 0,Y 383.062,Z 402.77,A -85,B 0,C 180,E1 -12130.716,E2 -12130.716} C_VEL
LIN {X 0,Y 383.083,Z 402.767,A -85,B 0,C 180,E1 -12134.026,E2 -12134.026} C_VEL
LIN {X 0,Y 383.138,Z 402.758,A -85,B 0,C 180,E1 -12137.284,E2 -12137.284} C_VEL
LIN {X 0,Y 383.153,Z 402.76,A -85,B 0,C 180,E1 -12140.498,E2 -12140.498} C_VEL
LIN {X 0,Y 383.276,Z 402.744,A -85,B 0,C 180,E1 -12142.625,E2 -12142.625} C_VEL
LIN {X 0,Y 383.2,Z 402.752,A -85,B 0,C 180,E1 -12144.738,E2 -12144.738} C_VEL
LIN {X 0,Y 383.387,Z 402.729,A -85,B 0,C 180,E1 -12147.899,E2 -12147.899} C_VEL
LIN {X 0,Y 383.52,Z 402.714,A -85,B 0,C 180,E1 -12150,E2 -12150} C_VEL
LIN {X 0,Y 383.252,Z 402.744,A -85,B 0,C 180,E1 -12153.153,E2 -12153.153} C_VEL
LIN {X 0,Y 383.206,Z 402.754,A -85,B 0,C 180,E1 -12156.317,E2 -12156.317} C_VEL
LIN {X 0,Y 382.744,Z 402.922,A -85,B 0,C 180,E1 -12159.512,E2 -12159.512} C_VEL
LIN {X 0,Y 382.583,Z 407.036,A -85,B 0,C 180,E1 -12163.193,E2 -12163.193} C_VEL
LIN {X 0,Y 382.298,Z 411.575,A -85,B 0,C 180,E1 -12167.105,E2 -12167.105} C_VEL
LIN {X 0,Y 382.065,Z 415.528,A -85,B 0,C 180,E1 -12170.456,E2 -12170.456} C_VEL
LIN {X 0,Y 381.94,Z 419.978,A -85,B 0,C 180,E1 -12174.168,E2 -12174.168} C_VEL
LIN {X 0,Y 381.947,Z 420.285,A -85,B 0,C 180,E1 -12174.42,E2 -12174.42} C_VEL
LIN {X 0,Y 385.158,Z 434.364,A -85,B 0,C 180,E1 -12175.102,E2 -12175.102} C_VEL
LIN {X 0,Y 387.404,Z 445.564,A -85,B 0,C 180,E1 -12175.81,E2 -12175.81} C_VEL
LIN {X 0,Y 387.389,Z 449.973,A -85,B 0,C 180,E1 -12176.1,E2 -12176.1} C_VEL
LIN {X 0,Y 386.533,Z 462.253,A -85,B 0,C 180,E1 -12177.036,E2 -12177.036} C_VEL
LIN {X 0,Y 386.223,Z 466.406,A -85,B 0,C 180,E1 -12177.417,E2 -12177.417} C_VEL
LIN {X 0,Y 385.273,Z 471.326,A -85,B 0,C 180,E1 -12177.882,E2 -12177.882} C_VEL
LIN {X 0,Y 381.835,Z 479.038,A -85,B 0,C 180,E1 -12178.661,E2 -12178.661} C_VEL
LIN {X 0,Y 378.344,Z 486.284,A -85,B 0,C 180,E1 -12179.541,E2 -12179.541} C_VEL
LIN {X 0,Y 377.323,Z 490.431,A -85,B 0,C 180,E1 -12180.158,E2 -12180.158} C_VEL
LIN {X 0,Y 376.449,Z 499.602,A -85,B 0,C 180,E1 -12181.813,E2 -12181.813} C_VEL
LIN {X 0,Y 375.773,Z 506.965,A -85,B 0,C 180,E1 -12183.485,E2 -12183.485} C_VEL
LIN {X 0,Y 375.315,Z 512.247,A -85,B 0,C 180,E1 -12184.981,E2 -12184.981} C_VEL
LIN {X 0,Y 374.9,Z 517.384,A -85,B 0,C 180,E1 -12186.861,E2 -12186.861} C_VEL
LIN {X 0,Y 374.701,Z 520.255,A -85,B 0,C 180,E1 -12188.239,E2 -12188.239} C_VEL
LIN {X 0,Y 374.459,Z 522.478,A -85,B 0,C 180,E1 -12189.691,E2 -12189.691} C_VEL
LIN {X 0,Y 374.365,Z 524.066,A -85,B 0,C 180,E1 -12191.329,E2 -12191.329} C_VEL
LIN {X 0,Y 374.357,Z 524.713,A -85,B 0,C 180,E1 -12192.931,E2 -12192.931} C_VEL
LIN {X 0,Y 374.363,Z 524.505,A -85,B 0,C 180,E1 -12194.489,E2 -12194.489} C_VEL
LIN {X 0,Y 374.445,Z 523.501,A -85,B 0,C 180,E1 -12196.016,E2 -12196.016} C_VEL
LIN {X 0,Y 374.652,Z 521.714,A -85,B 0,C 180,E1 -12197.521,E2 -12197.521} C_VEL
LIN {X 0,Y 374.94,Z 519.117,A -85,B 0,C 180,E1 -12199.001,E2 -12199.001} C_VEL
LIN {X 0,Y 375.239,Z 515.766,A -85,B 0,C 180,E1 -12200.446,E2 -12200.446} C_VEL
LIN {X 0,Y 375.796,Z 510.404,A -85,B 0,C 180,E1 -12202.231,E2 -12202.231} C_VEL
LIN {X 0,Y 376.546,Z 503.264,A -85,B 0,C 180,E1 -12204.059,E2 -12204.059} C_VEL
LIN {X 0,Y 377.355,Z 495.813,A -85,B 0,C 180,E1 -12205.574,E2 -12205.574} C_VEL
LIN {X 0,Y 378.4,Z 486.566,A -85,B 0,C 180,E1 -12207.097,E2 -12207.097} C_VEL
LIN {X 0,Y 379.48,Z 476.547,A -85,B 0,C 180,E1 -12208.42,E2 -12208.42} C_VEL
LIN {X 0,Y 380.517,Z 465.098,A -85,B 0,C 180,E1 -12209.629,E2 -12209.629} C_VEL
LIN {X 0,Y 381.467,Z 453.051,A -85,B 0,C 180,E1 -12210.625,E2 -12210.625} C_VEL
LIN {X 0,Y 381.719,Z 448.664,A -85,B 0,C 180,E1 -12210.929,E2 -12210.929} C_VEL
LIN {X 0,Y 379.608,Z 438.189,A -85,B 0,C 180,E1 -12211.691,E2 -12211.691} C_VEL
LIN {X 0,Y 376.31,Z 426.044,A -85,B 0,C 180,E1 -12212.431,E2 -12212.431} C_VEL
LIN {X 0,Y 375.078,Z 421.724,A -85,B 0,C 180,E1 -12212.673,E2 -12212.673} C_VEL
LIN {X 0,Y 375.249,Z 418.417,A -85,B 0,C 180,E1 -12215.667,E2 -12215.667} C_VEL
LIN {X 0,Y 375.404,Z 415.875,A -85,B 0,C 180,E1 -12218.011,E2 -12218.011} C_VEL
LIN {X 0,Y 375.675,Z 412.244,A -85,B 0,C 180,E1 -12221.456,E2 -12221.456} C_VEL
LIN {X 0,Y 375.941,Z 408.832,A -85,B 0,C 180,E1 -12224.828,E2 -12224.828} C_VEL
LIN {X 0,Y 376.121,Z 406.643,A -85,B 0,C 180,E1 -12227.043,E2 -12227.043} C_VEL
LIN {X 0,Y 376.071,Z 403.647,A -85,B 0,C 180,E1 -12230.317,E2 -12230.317} C_VEL
LIN {X 0,Y 376.227,Z 403.625,A -85,B 0,C 180,E1 -12232.486,E2 -12232.486} C_VEL
LIN {X 0,Y 376.168,Z 403.63,A -85,B 0,C 180,E1 -12234.64,E2 -12234.64} C_VEL
LIN {X 0,Y 376.35,Z 403.61,A -85,B 0,C 180,E1 -12237.86,E2 -12237.86} C_VEL
LIN {X 0,Y 376.487,Z 403.59,A -85,B 0,C 180,E1 -12240,E2 -12240} C_VEL
LIN {X 0,Y 376.186,Z 403.628,A -85,B 0,C 180,E1 -12243.213,E2 -12243.213} C_VEL
LIN {X 0,Y 376.243,Z 403.621,A -85,B 0,C 180,E1 -12246.435,E2 -12246.435} C_VEL
LIN {X 0,Y 376.201,Z 403.626,A -85,B 0,C 180,E1 -12248.595,E2 -12248.595} C_VEL
LIN {X 0,Y 376.046,Z 403.645,A -85,B 0,C 180,E1 -12251.864,E2 -12251.864} C_VEL
LIN {X 0,Y 376.054,Z 403.644,A -85,B 0,C 180,E1 -12255.168,E2 -12255.168} C_VEL
LIN {X 0,Y 376.02,Z 403.648,A -85,B 0,C 180,E1 -12258.526,E2 -12258.526} C_VEL
LIN {X 0,Y 375.959,Z 403.655,A -85,B 0,C 180,E1 -12261.955,E2 -12261.955} C_VEL
LIN {X 0,Y 376.003,Z 403.651,A -85,B 0,C 180,E1 -12265.461,E2 -12265.461} C_VEL
LIN {X 0,Y 375.973,Z 403.654,A -85,B 0,C 180,E1 -12269.079,E2 -12269.079} C_VEL
LIN {X 0,Y 375.948,Z 403.658,A -85,B 0,C 180,E1 -12272.829,E2 -12272.829} C_VEL
LIN {X 0,Y 375.956,Z 403.658,A -85,B 0,C 180,E1 -12275.416,E2 -12275.416} C_VEL
LIN {X 0,Y 375.976,Z 403.657,A -85,B 0,C 180,E1 -12278.272,E2 -12278.272} C_VEL
LIN {X 0,Y 375.958,Z 403.659,A -85,B 0,C 180,E1 -12281.606,E2 -12281.606} C_VEL
LIN {X 0,Y 375.994,Z 403.795,A -85,B 0,C 180,E1 -12285.259,E2 -12285.259} C_VEL
LIN {X 0,Y 376.892,Z 408.892,A -85,B 0,C 180,E1 -12289.259,E2 -12289.259} C_VEL
LIN {X 0,Y 377.524,Z 412.918,A -85,B 0,C 180,E1 -12292.098,E2 -12292.098} C_VEL
LIN {X 0,Y 377.723,Z 416.033,A -85,B 0,C 180,E1 -12294.12,E2 -12294.12} C_VEL
LIN {X 0,Y 377.276,Z 420.737,A -85,B 0,C 180,E1 -12296.959,E2 -12296.959} C_VEL
LIN {X 0,Y 376.631,Z 426.698,A -85,B 0,C 180,E1 -12300.364,E2 -12300.364} C_VEL
LIN {X 0,Y 376.078,Z 432.936,A -85,B 0,C 180,E1 -12303.768,E2 -12303.768} C_VEL
LIN {X 0,Y 375.606,Z 439.965,A -85,B 0,C 180,E1 -12307.445,E2 -12307.445} C_VEL
LIN {X 0,Y 375.222,Z 445.763,A -85,B 0,C 180,E1 -12310.351,E2 -12310.351} C_VEL
LIN {X 0,Y 378.045,Z 459.094,A -85,B 0,C 180,E1 -12310.998,E2 -12310.998} C_VEL
LIN {X 0,Y 379.652,Z 469.974,A -85,B 0,C 180,E1 -12311.658,E2 -12311.658} C_VEL
LIN {X 0,Y 380.56,Z 482.323,A -85,B 0,C 180,E1 -12312.565,E2 -12312.565} C_VEL
LIN {X 0,Y 379.494,Z 494.404,A -85,B 0,C 180,E1 -12313.596,E2 -12313.596} C_VEL
LIN {X 0,Y 378.343,Z 505.443,A -85,B 0,C 180,E1 -12314.789,E2 -12314.789} C_VEL
LIN {X 0,Y 377.484,Z 514.454,A -85,B 0,C 180,E1 -12315.994,E2 -12315.994} C_VEL
LIN {X 0,Y 376.533,Z 524.261,A -85,B 0,C 180,E1 -12317.606,E2 -12317.606} C_VEL
LIN {X 0,Y 375.668,Z 532.138,A -85,B 0,C 180,E1 -12319.218,E2 -12319.218} C_VEL
LIN {X 0,Y 375.18,Z 538.466,A -85,B 0,C 180,E1 -12320.839,E2 -12320.839} C_VEL
LIN {X 0,Y 374.796,Z 543.516,A -85,B 0,C 180,E1 -12322.458,E2 -12322.458} C_VEL
LIN {X 0,Y 374.59,Z 547.122,A -85,B 0,C 180,E1 -12323.924,E2 -12323.924} C_VEL
LIN {X 0,Y 374.555,Z 550.321,A -85,B 0,C 180,E1 -12325.696,E2 -12325.696} C_VEL
LIN {X 0,Y 374.499,Z 552.668,A -85,B 0,C 180,E1 -12327.849,E2 -12327.849} C_VEL
LIN {X 0,Y 374.584,Z 553.246,A -85,B 0,C 180,E1 -12328.925,E2 -12328.925} C_VEL
LIN {X 0,Y 374.589,Z 553.38,A -85,B 0,C 180,E1 -12330,E2 -12330} C_VEL
LIN {X 0,Y 374.586,Z 553.115,A -85,B 0,C 180,E1 -12331.075,E2 -12331.075} C_VEL
LIN {X 0,Y 374.519,Z 552.456,A -85,B 0,C 180,E1 -12332.151,E2 -12332.151} C_VEL
LIN {X 0,Y 374.477,Z 551.394,A -85,B 0,C 180,E1 -12333.228,E2 -12333.228} C_VEL
LIN {X 0,Y 374.559,Z 549.875,A -85,B 0,C 180,E1 -12334.305,E2 -12334.305} C_VEL
LIN {X 0,Y 374.586,Z 546.446,A -85,B 0,C 180,E1 -12336.071,E2 -12336.071} C_VEL
LIN {X 0,Y 374.881,Z 541,A -85,B 0,C 180,E1 -12338.083,E2 -12338.083} C_VEL
LIN {X 0,Y 375.353,Z 534.105,A -85,B 0,C 180,E1 -12339.974,E2 -12339.974} C_VEL
LIN {X 0,Y 375.955,Z 526.618,A -85,B 0,C 180,E1 -12341.593,E2 -12341.593} C_VEL
LIN {X 0,Y 376.717,Z 518.993,A -85,B 0,C 180,E1 -12342.937,E2 -12342.937} C_VEL
LIN {X 0,Y 377.512,Z 510.306,A -85,B 0,C 180,E1 -12344.205,E2 -12344.205} C_VEL
LIN {X 0,Y 378.271,Z 500.764,A -85,B 0,C 180,E1 -12345.353,E2 -12345.353} C_VEL
LIN {X 0,Y 379.223,Z 489.722,A -85,B 0,C 180,E1 -12346.417,E2 -12346.417} C_VEL
LIN {X 0,Y 379.84,Z 479.372,A -85,B 0,C 180,E1 -12347.22,E2 -12347.22} C_VEL
LIN {X 0,Y 378.313,Z 466.091,A -85,B 0,C 180,E1 -12348.098,E2 -12348.098} C_VEL
LIN {X 0,Y 376.205,Z 452.904,A -85,B 0,C 180,E1 -12348.754,E2 -12348.754} C_VEL
LIN {X 0,Y 375.123,Z 446.804,A -85,B 0,C 180,E1 -12348.998,E2 -12348.998} C_VEL
LIN {X 0,Y 375.503,Z 440.843,A -85,B 0,C 180,E1 -12351.983,E2 -12351.983} C_VEL
LIN {X 0,Y 375.898,Z 434.011,A -85,B 0,C 180,E1 -12355.469,E2 -12355.469} C_VEL
LIN {X 0,Y 376.475,Z 427.192,A -85,B 0,C 180,E1 -12359.037,E2 -12359.037} C_VEL
LIN {X 0,Y 376.961,Z 421.494,A -85,B 0,C 180,E1 -12362.097,E2 -12362.097} C_VEL
LIN {X 0,Y 377.545,Z 415.801,A -85,B 0,C 180,E1 -12365.245,E2 -12365.245} C_VEL
LIN {X 0,Y 377.246,Z 411.212,A -85,B 0,C 180,E1 -12367.936,E2 -12367.936} C_VEL
LIN {X 0,Y 376.511,Z 406.611,A -85,B 0,C 180,E1 -12370.792,E2 -12370.792} C_VEL
LIN {X 0,Y 376.009,Z 403.65,A -85,B 0,C 180,E1 -12372.736,E2 -12372.736} C_VEL
LIN {X 0,Y 375.935,Z 403.657,A -85,B 0,C 180,E1 -12376.811,E2 -12376.811} C_VEL
LIN {X 0,Y 375.963,Z 403.652,A -85,B 0,C 180,E1 -12380.537,E2 -12380.537} C_VEL
LIN {X 0,Y 375.965,Z 403.655,A -85,B 0,C 180,E1 -12383.495,E2 -12383.495} C_VEL
LIN {X 0,Y 375.961,Z 403.652,A -85,B 0,C 180,E1 -12385.888,E2 -12385.888} C_VEL
LIN {X 0,Y 375.966,Z 403.653,A -85,B 0,C 180,E1 -12389.687,E2 -12389.687} C_VEL
LIN {X 0,Y 376.021,Z 403.648,A -85,B 0,C 180,E1 -12393.348,E2 -12393.348} C_VEL
LIN {X 0,Y 375.998,Z 403.651,A -85,B 0,C 180,E1 -12396.888,E2 -12396.888} C_VEL
LIN {X 0,Y 375.999,Z 403.647,A -85,B 0,C 180,E1 -12400.339,E2 -12400.339} C_VEL
LIN {X 0,Y 376.029,Z 403.644,A -85,B 0,C 180,E1 -12403.719,E2 -12403.719} C_VEL
LIN {X 0,Y 376.104,Z 403.639,A -85,B 0,C 180,E1 -12407.042,E2 -12407.042} C_VEL
LIN {X 0,Y 376.12,Z 403.632,A -85,B 0,C 180,E1 -12410.318,E2 -12410.318} C_VEL
LIN {X 0,Y 376.231,Z 403.62,A -85,B 0,C 180,E1 -12412.486,E2 -12412.486} C_VEL
LIN {X 0,Y 376.171,Z 403.629,A -85,B 0,C 180,E1 -12414.64,E2 -12414.64} C_VEL
LIN {X 0,Y 376.352,Z 403.603,A -85,B 0,C 180,E1 -12417.86,E2 -12417.86} C_VEL
LIN {X 0,Y 376.487,Z 403.586,A -85,B 0,C 180,E1 -12420,E2 -12420} C_VEL
LIN {X 0,Y 376.185,Z 403.627,A -85,B 0,C 180,E1 -12423.213,E2 -12423.213} C_VEL
LIN {X 0,Y 376.235,Z 403.618,A -85,B 0,C 180,E1 -12426.62,E2 -12426.62} C_VEL
LIN {X 0,Y 376.206,Z 403.624,A -85,B 0,C 180,E1 -12428.595,E2 -12428.595} C_VEL
LIN {X 0,Y 376.05,Z 403.641,A -85,B 0,C 180,E1 -12431.863,E2 -12431.863} C_VEL
LIN {X 0,Y 376.059,Z 403.643,A -85,B 0,C 180,E1 -12435.167,E2 -12435.167} C_VEL
LIN {X 0,Y 376.025,Z 403.647,A -85,B 0,C 180,E1 -12438.526,E2 -12438.526} C_VEL
LIN {X 0,Y 375.964,Z 403.651,A -85,B 0,C 180,E1 -12441.954,E2 -12441.954} C_VEL
LIN {X 0,Y 376.007,Z 403.646,A -85,B 0,C 180,E1 -12445.461,E2 -12445.461} C_VEL
LIN {X 0,Y 375.971,Z 403.654,A -85,B 0,C 180,E1 -12449.079,E2 -12449.079} C_VEL
LIN {X 0,Y 375.95,Z 403.657,A -85,B 0,C 180,E1 -12452.828,E2 -12452.828} C_VEL
LIN {X 0,Y 375.958,Z 403.653,A -85,B 0,C 180,E1 -12455.415,E2 -12455.415} C_VEL
LIN {X 0,Y 375.974,Z 403.652,A -85,B 0,C 180,E1 -12458.27,E2 -12458.27} C_VEL
LIN {X 0,Y 375.935,Z 403.655,A -85,B 0,C 180,E1 -12461.601,E2 -12461.601} C_VEL
LIN {X 0,Y 375.928,Z 403.657,A -85,B 0,C 180,E1 -12465.269,E2 -12465.269} C_VEL
LIN {X 0,Y 375.936,Z 403.659,A -85,B 0,C 180,E1 -12468.399,E2 -12468.399} C_VEL
LIN {X 0,Y 375.976,Z 403.65,A -85,B 0,C 180,E1 -12471.729,E2 -12471.729} C_VEL
LIN {X 0,Y 375.981,Z 403.649,A -85,B 0,C 180,E1 -12475.333,E2 -12475.333} C_VEL
LIN {X 0,Y 375.959,Z 403.656,A -85,B 0,C 180,E1 -12478.438,E2 -12478.438} C_VEL
LIN {X 0,Y 375.985,Z 403.651,A -85,B 0,C 180,E1 -12482.14,E2 -12482.14} C_VEL
LIN {X 0,Y 376.009,Z 403.65,A -85,B 0,C 180,E1 -12484.539,E2 -12484.539} C_VEL
LIN {X 0,Y 375.965,Z 403.653,A -85,B 0,C 180,E1 -12488.046,E2 -12488.046} C_VEL
LIN {X 0,Y 376.011,Z 403.645,A -85,B 0,C 180,E1 -12491.473,E2 -12491.473} C_VEL
LIN {X 0,Y 376.06,Z 403.642,A -85,B 0,C 180,E1 -12494.832,E2 -12494.832} C_VEL
LIN {X 0,Y 376.052,Z 403.644,A -85,B 0,C 180,E1 -12498.136,E2 -12498.136} C_VEL
LIN {X 0,Y 376.26,Z 403.616,A -85,B 0,C 180,E1 -12501.877,E2 -12501.877} C_VEL
LIN {X 0,Y 376.173,Z 403.628,A -85,B 0,C 180,E1 -12504.64,E2 -12504.64} C_VEL
LIN {X 0,Y 376.353,Z 403.605,A -85,B 0,C 180,E1 -12507.859,E2 -12507.859} C_VEL
LIN {X 0,Y 376.489,Z 403.589,A -85,B 0,C 180,E1 -12510,E2 -12510} C_VEL
LIN {X 0,Y 376.19,Z 403.623,A -85,B 0,C 180,E1 -12513.212,E2 -12513.212} C_VEL
LIN {X 0,Y 376.155,Z 403.632,A -85,B 0,C 180,E1 -12516.436,E2 -12516.436} C_VEL
LIN {X 0,Y 375.837,Z 403.671,A -85,B 0,C 180,E1 -12518.603,E2 -12518.603} C_VEL
LIN {X 0,Y 375.695,Z 403.978,A -85,B 0,C 180,E1 -12519.692,E2 -12519.692} C_VEL
LIN {X 0,Y 375.538,Z 407.977,A -85,B 0,C 180,E1 -12523.306,E2 -12523.306} C_VEL
LIN {X 0,Y 375.232,Z 412.441,A -85,B 0,C 180,E1 -12527.212,E2 -12527.212} C_VEL
LIN {X 0,Y 374.969,Z 416.74,A -85,B 0,C 180,E1 -12530.861,E2 -12530.861} C_VEL
LIN {X 0,Y 374.897,Z 420.552,A -85,B 0,C 180,E1 -12534.099,E2 -12534.099} C_VEL
LIN {X 0,Y 378.119,Z 434.561,A -85,B 0,C 180,E1 -12534.794,E2 -12534.794} C_VEL
LIN {X 0,Y 380.523,Z 446.6,A -85,B 0,C 180,E1 -12535.576,E2 -12535.576} C_VEL
LIN {X 0,Y 380.501,Z 450.917,A -85,B 0,C 180,E1 -12535.871,E2 -12535.871} C_VEL
LIN {X 0,Y 379.65,Z 462.535,A -85,B 0,C 180,E1 -12536.779,E2 -12536.779} C_VEL
LIN {X 0,Y 378.773,Z 473.995,A -85,B 0,C 180,E1 -12537.937,E2 -12537.937} C_VEL
LIN {X 0,Y 377.789,Z 484.723,A -85,B 0,C 180,E1 -12539.29,E2 -12539.29} C_VEL
LIN {X 0,Y 377.323,Z 490.431,A -85,B 0,C 180,E1 -12540.158,E2 -12540.158} C_VEL
LIN {X 0,Y 376.324,Z 494.424,A -85,B 0,C 180,E1 -12540.806,E2 -12540.806} C_VEL
LIN {X 0,Y 372.902,Z 500.518,A -85,B 0,C 180,E1 -12541.886,E2 -12541.886} C_VEL
LIN {X 0,Y 369.513,Z 506.007,A -85,B 0,C 180,E1 -12543.052,E2 -12543.052} C_VEL
LIN {X 0,Y 368.579,Z 509.016,A -85,B 0,C 180,E1 -12543.824,E2 -12543.824} C_VEL
LIN {X 0,Y 368.086,Z 514.723,A -85,B 0,C 180,E1 -12545.615,E2 -12545.615} C_VEL
LIN {X 0,Y 367.666,Z 519.629,A -85,B 0,C 180,E1 -12547.711,E2 -12547.711} C_VEL
LIN {X 0,Y 367.462,Z 522.034,A -85,B 0,C 180,E1 -12549.134,E2 -12549.134} C_VEL
LIN {X 0,Y 367.29,Z 523.754,A -85,B 0,C 180,E1 -12550.584,E2 -12550.584} C_VEL
LIN {X 0,Y 367.26,Z 524.727,A -85,B 0,C 180,E1 -12552.048,E2 -12552.048} C_VEL
LIN {X 0,Y 367.252,Z 525.014,A -85,B 0,C 180,E1 -12553.544,E2 -12553.544} C_VEL
LIN {X 0,Y 367.3,Z 524.56,A -85,B 0,C 180,E1 -12555.069,E2 -12555.069} C_VEL
LIN {X 0,Y 367.436,Z 523.268,A -85,B 0,C 180,E1 -12556.62,E2 -12556.62} C_VEL
LIN {X 0,Y 367.707,Z 521.12,A -85,B 0,C 180,E1 -12558.193,E2 -12558.193} C_VEL
LIN {X 0,Y 368.035,Z 518.009,A -85,B 0,C 180,E1 -12559.803,E2 -12559.803} C_VEL
LIN {X 0,Y 368.457,Z 513.79,A -85,B 0,C 180,E1 -12561.446,E2 -12561.446} C_VEL
LIN {X 0,Y 369.096,Z 508.349,A -85,B 0,C 180,E1 -12563.103,E2 -12563.103} C_VEL
LIN {X 0,Y 369.884,Z 501.416,A -85,B 0,C 180,E1 -12564.787,E2 -12564.787} C_VEL
LIN {X 0,Y 370.76,Z 493.881,A -85,B 0,C 180,E1 -12566.26,E2 -12566.26} C_VEL
LIN {X 0,Y 371.837,Z 484.61,A -85,B 0,C 180,E1 -12567.728,E2 -12567.728} C_VEL
LIN {X 0,Y 373.003,Z 473.799,A -85,B 0,C 180,E1 -12569.107,E2 -12569.107} C_VEL
LIN {X 0,Y 373.987,Z 463.242,A -85,B 0,C 180,E1 -12570.181,E2 -12570.181} C_VEL
LIN {X 0,Y 374.985,Z 451.135,A -85,B 0,C 180,E1 -12571.144,E2 -12571.144} C_VEL
LIN {X 0,Y 373.621,Z 442.691,A -85,B 0,C 180,E1 -12571.796,E2 -12571.796} C_VEL
LIN {X 0,Y 370.325,Z 429.564,A -85,B 0,C 180,E1 -12572.676,E2 -12572.676} C_VEL
LIN {X 0,Y 368.055,Z 422.02,A -85,B 0,C 180,E1 -12573.136,E2 -12573.136} C_VEL
LIN {X 0,Y 368.274,Z 418.51,A -85,B 0,C 180,E1 -12576.375,E2 -12576.375} C_VEL
LIN {X 0,Y 368.509,Z 414.795,A -85,B 0,C 180,E1 -12579.923,E2 -12579.923} C_VEL
LIN {X 0,Y 368.775,Z 411.286,A -85,B 0,C 180,E1 -12583.389,E2 -12583.389} C_VEL
LIN {X 0,Y 369.083,Z 407.975,A -85,B 0,C 180,E1 -12586.791,E2 -12586.791} C_VEL
LIN {X 0,Y 369.07,Z 404.908,A -85,B 0,C 180,E1 -12590.132,E2 -12590.132} C_VEL
LIN {X 0,Y 369.205,Z 404.501,A -85,B 0,C 180,E1 -12591.822,E2 -12591.822} C_VEL
LIN {X 0,Y 369.141,Z 404.506,A -85,B 0,C 180,E1 -12594.538,E2 -12594.538} C_VEL
LIN {X 0,Y 369.315,Z 404.486,A -85,B 0,C 180,E1 -12597.819,E2 -12597.819} C_VEL
LIN {X 0,Y 369.456,Z 404.466,A -85,B 0,C 180,E1 -12600,E2 -12600} C_VEL
LIN {X 0,Y 369.315,Z 404.481,A -85,B 0,C 180,E1 -12602.181,E2 -12602.181} C_VEL
LIN {X 0,Y 369.204,Z 404.497,A -85,B 0,C 180,E1 -12606.558,E2 -12606.558} C_VEL
LIN {X 0,Y 369.133,Z 404.506,A -85,B 0,C 180,E1 -12608.761,E2 -12608.761} C_VEL
LIN {X 0,Y 369.001,Z 404.522,A -85,B 0,C 180,E1 -12612.094,E2 -12612.094} C_VEL
LIN {X 0,Y 368.994,Z 404.524,A -85,B 0,C 180,E1 -12615.465,E2 -12615.465} C_VEL
LIN {X 0,Y 368.979,Z 404.525,A -85,B 0,C 180,E1 -12618.893,E2 -12618.893} C_VEL
LIN {X 0,Y 368.929,Z 404.531,A -85,B 0,C 180,E1 -12622.395,E2 -12622.395} C_VEL
LIN {X 0,Y 368.996,Z 404.523,A -85,B 0,C 180,E1 -12625.981,E2 -12625.981} C_VEL
LIN {X 0,Y 368.964,Z 404.528,A -85,B 0,C 180,E1 -12628.814,E2 -12628.814} C_VEL
LIN {X 0,Y 368.897,Z 404.536,A -85,B 0,C 180,E1 -12632.238,E2 -12632.238} C_VEL
LIN {X 0,Y 368.927,Z 404.534,A -85,B 0,C 180,E1 -12635.002,E2 -12635.002} C_VEL
LIN {X 0,Y 368.911,Z 404.537,A -85,B 0,C 180,E1 -12638.642,E2 -12638.642} C_VEL
LIN {X 0,Y 368.908,Z 404.537,A -85,B 0,C 180,E1 -12641.819,E2 -12641.819} C_VEL
LIN {X 0,Y 368.992,Z 404.735,A -85,B 0,C 180,E1 -12644.807,E2 -12644.807} C_VEL
LIN {X 0,Y 369.702,Z 409.01,A -85,B 0,C 180,E1 -12648.292,E2 -12648.292} C_VEL
LIN {X 0,Y 370.343,Z 412.983,A -85,B 0,C 180,E1 -12651.228,E2 -12651.228} C_VEL
LIN {X 0,Y 370.658,Z 415.21,A -85,B 0,C 180,E1 -12652.784,E2 -12652.784} C_VEL
LIN {X 0,Y 370.604,Z 419.153,A -85,B 0,C 180,E1 -12655.327,E2 -12655.327} C_VEL
LIN {X 0,Y 369.835,Z 425.551,A -85,B 0,C 180,E1 -12659.131,E2 -12659.131} C_VEL
LIN {X 0,Y 369.162,Z 432.066,A -85,B 0,C 180,E1 -12662.813,E2 -12662.813} C_VEL
LIN {X 0,Y 368.646,Z 438.689,A -85,B 0,C 180,E1 -12666.401,E2 -12666.401} C_VEL
LIN {X 0,Y 368.205,Z 445.237,A -85,B 0,C 180,E1 -12669.823,E2 -12669.823} C_VEL
LIN {X 0,Y 368.213,Z 445.565,A -85,B 0,C 180,E1 -12669.907,E2 -12669.907} C_VEL
LIN {X 0,Y 371.232,Z 459.549,A -85,B 0,C 180,E1 -12670.624,E2 -12670.624} C_VEL
LIN {X 0,Y 372.957,Z 471.423,A -85,B 0,C 180,E1 -12671.384,E2 -12671.384} C_VEL
LIN {X 0,Y 373.777,Z 482.599,A -85,B 0,C 180,E1 -12672.24,E2 -12672.24} C_VEL
LIN {X 0,Y 372.69,Z 494.55,A -85,B 0,C 180,E1 -12673.288,E2 -12673.288} C_VEL
LIN {X 0,Y 371.487,Z 505.476,A -85,B 0,C 180,E1 -12674.501,E2 -12674.501} C_VEL
LIN {X 0,Y 370.551,Z 514.416,A -85,B 0,C 180,E1 -12675.726,E2 -12675.726} C_VEL
LIN {X 0,Y 369.721,Z 522.666,A -85,B 0,C 180,E1 -12677.094,E2 -12677.094} C_VEL
LIN {X 0,Y 368.777,Z 530.788,A -85,B 0,C 180,E1 -12678.736,E2 -12678.736} C_VEL
LIN {X 0,Y 368.278,Z 536.334,A -85,B 0,C 180,E1 -12680.111,E2 -12680.111} C_VEL
LIN {X 0,Y 367.843,Z 541.779,A -85,B 0,C 180,E1 -12681.762,E2 -12681.762} C_VEL
LIN {X 0,Y 367.564,Z 546.042,A -85,B 0,C 180,E1 -12683.413,E2 -12683.413} C_VEL
LIN {X 0,Y 367.47,Z 548.309,A -85,B 0,C 180,E1 -12684.513,E2 -12684.513} C_VEL
LIN {X 0,Y 367.46,Z 550.088,A -85,B 0,C 180,E1 -12685.613,E2 -12685.613} C_VEL
LIN {X 0,Y 367.399,Z 552.418,A -85,B 0,C 180,E1 -12687.808,E2 -12687.808} C_VEL
LIN {X 0,Y 367.484,Z 552.981,A -85,B 0,C 180,E1 -12688.905,E2 -12688.905} C_VEL
LIN {X 0,Y 367.505,Z 553.101,A -85,B 0,C 180,E1 -12690,E2 -12690} C_VEL
LIN {X 0,Y 367.487,Z 552.825,A -85,B 0,C 180,E1 -12691.096,E2 -12691.096} C_VEL
LIN {X 0,Y 367.419,Z 552.156,A -85,B 0,C 180,E1 -12692.193,E2 -12692.193} C_VEL
LIN {X 0,Y 367.394,Z 551.077,A -85,B 0,C 180,E1 -12693.29,E2 -12693.29} C_VEL
LIN {X 0,Y 367.464,Z 549.54,A -85,B 0,C 180,E1 -12694.388,E2 -12694.388} C_VEL
LIN {X 0,Y 367.484,Z 546.468,A -85,B 0,C 180,E1 -12696.02,E2 -12696.02} C_VEL
LIN {X 0,Y 367.708,Z 542.241,A -85,B 0,C 180,E1 -12697.689,E2 -12697.689} C_VEL
LIN {X 0,Y 368.156,Z 535.844,A -85,B 0,C 180,E1 -12699.616,E2 -12699.616} C_VEL
LIN {X 0,Y 368.708,Z 528.865,A -85,B 0,C 180,E1 -12701.267,E2 -12701.267} C_VEL
LIN {X 0,Y 369.616,Z 520.121,A -85,B 0,C 180,E1 -12702.91,E2 -12702.91} C_VEL
LIN {X 0,Y 370.543,Z 510.178,A -85,B 0,C 180,E1 -12704.417,E2 -12704.417} C_VEL
LIN {X 0,Y 371.389,Z 500.123,A -85,B 0,C 180,E1 -12705.644,E2 -12705.644} C_VEL
LIN {X 0,Y 372.387,Z 488.995,A -85,B 0,C 180,E1 -12706.727,E2 -12706.727} C_VEL
LIN {X 0,Y 372.932,Z 480.5,A -85,B 0,C 180,E1 -12707.408,E2 -12707.408} C_VEL
LIN {X 0,Y 371.621,Z 468.306,A -85,B 0,C 180,E1 -12708.257,E2 -12708.257} C_VEL
LIN {X 0,Y 369.667,Z 455.601,A -85,B 0,C 180,E1 -12708.951,E2 -12708.951} C_VEL
LIN {X 0,Y 368.089,Z 446.531,A -85,B 0,C 180,E1 -12709.339,E2 -12709.339} C_VEL
LIN {X 0,Y 368.456,Z 440.529,A -85,B 0,C 180,E1 -12712.426,E2 -12712.426} C_VEL
LIN {X 0,Y 368.977,Z 432.812,A -85,B 0,C 180,E1 -12716.463,E2 -12716.463} C_VEL
LIN {X 0,Y 369.633,Z 425.76,A -85,B 0,C 180,E1 -12720.256,E2 -12720.256} C_VEL
LIN {X 0,Y 370.301,Z 418.944,A -85,B 0,C 180,E1 -12724.048,E2 -12724.048} C_VEL
LIN {X 0,Y 370.495,Z 415.511,A -85,B 0,C 180,E1 -12726.019,E2 -12726.019} C_VEL
LIN {X 0,Y 370.052,Z 410.833,A -85,B 0,C 180,E1 -12728.861,E2 -12728.861} C_VEL
LIN {X 0,Y 369.187,Z 405.868,A -85,B 0,C 180,E1 -12732.062,E2 -12732.062} C_VEL
LIN {X 0,Y 368.944,Z 404.53,A -85,B 0,C 180,E1 -12733.056,E2 -12733.056} C_VEL
LIN {X 0,Y 368.887,Z 404.535,A -85,B 0,C 180,E1 -12736.696,E2 -12736.696} C_VEL
LIN {X 0,Y 368.912,Z 404.532,A -85,B 0,C 180,E1 -12739.643,E2 -12739.643} C_VEL
LIN {X 0,Y 368.902,Z 404.536,A -85,B 0,C 180,E1 -12743.144,E2 -12743.144} C_VEL
LIN {X 0,Y 368.897,Z 404.532,A -85,B 0,C 180,E1 -12746.462,E2 -12746.462} C_VEL
LIN {X 0,Y 368.93,Z 404.532,A -85,B 0,C 180,E1 -12749.046,E2 -12749.046} C_VEL
LIN {X 0,Y 368.977,Z 404.524,A -85,B 0,C 180,E1 -12751.564,E2 -12751.564} C_VEL
LIN {X 0,Y 369.001,Z 404.518,A -85,B 0,C 180,E1 -12754.02,E2 -12754.02} C_VEL
LIN {X 0,Y 368.933,Z 404.528,A -85,B 0,C 180,E1 -12757.605,E2 -12757.605} C_VEL
LIN {X 0,Y 368.959,Z 404.529,A -85,B 0,C 180,E1 -12761.106,E2 -12761.106} C_VEL
LIN {X 0,Y 368.998,Z 404.52,A -85,B 0,C 180,E1 -12764.535,E2 -12764.535} C_VEL
LIN {X 0,Y 369.006,Z 404.518,A -85,B 0,C 180,E1 -12767.907,E2 -12767.907} C_VEL
LIN {X 0,Y 369.23,Z 404.49,A -85,B 0,C 180,E1 -12771.801,E2 -12771.801} C_VEL
LIN {X 0,Y 369.144,Z 404.503,A -85,B 0,C 180,E1 -12774.537,E2 -12774.537} C_VEL
LIN {X 0,Y 369.317,Z 404.479,A -85,B 0,C 180,E1 -12777.819,E2 -12777.819} C_VEL
LIN {X 0,Y 369.457,Z 404.462,A -85,B 0,C 180,E1 -12780,E2 -12780} C_VEL
LIN {X 0,Y 369.317,Z 404.479,A -85,B 0,C 180,E1 -12782.181,E2 -12782.181} C_VEL
LIN {X 0,Y 369.205,Z 404.496,A -85,B 0,C 180,E1 -12786.607,E2 -12786.607} C_VEL
LIN {X 0,Y 369.139,Z 404.506,A -85,B 0,C 180,E1 -12788.761,E2 -12788.761} C_VEL
LIN {X 0,Y 369.005,Z 404.518,A -85,B 0,C 180,E1 -12792.093,E2 -12792.093} C_VEL
LIN {X 0,Y 368.998,Z 404.52,A -85,B 0,C 180,E1 -12795.465,E2 -12795.465} C_VEL
LIN {X 0,Y 368.983,Z 404.526,A -85,B 0,C 180,E1 -12798.893,E2 -12798.893} C_VEL
LIN {X 0,Y 368.933,Z 404.529,A -85,B 0,C 180,E1 -12802.395,E2 -12802.395} C_VEL
LIN {X 0,Y 369.001,Z 404.518,A -85,B 0,C 180,E1 -12805.98,E2 -12805.98} C_VEL
LIN {X 0,Y 368.962,Z 404.528,A -85,B 0,C 180,E1 -12808.811,E2 -12808.811} C_VEL
LIN {X 0,Y 368.899,Z 404.533,A -85,B 0,C 180,E1 -12812.238,E2 -12812.238} C_VEL
LIN {X 0,Y 368.93,Z 404.531,A -85,B 0,C 180,E1 -12815.001,E2 -12815.001} C_VEL
LIN {X 0,Y 368.909,Z 404.535,A -85,B 0,C 180,E1 -12818.64,E2 -12818.64} C_VEL
LIN {X 0,Y 368.882,Z 404.534,A -85,B 0,C 180,E1 -12822.009,E2 -12822.009} C_VEL
LIN {X 0,Y 368.88,Z 404.535,A -85,B 0,C 180,E1 -12825.176,E2 -12825.176} C_VEL
LIN {X 0,Y 368.884,Z 404.535,A -85,B 0,C 180,E1 -12828.178,E2 -12828.178} C_VEL
LIN {X 0,Y 368.911,Z 404.53,A -85,B 0,C 180,E1 -12831.359,E2 -12831.359} C_VEL
LIN {X 0,Y 368.938,Z 404.527,A -85,B 0,C 180,E1 -12835.146,E2 -12835.146} C_VEL
LIN {X 0,Y 368.931,Z 404.529,A -85,B 0,C 180,E1 -12839.046,E2 -12839.046} C_VEL
LIN {X 0,Y 368.965,Z 404.526,A -85,B 0,C 180,E1 -12842.796,E2 -12842.796} C_VEL
LIN {X 0,Y 368.947,Z 404.528,A -85,B 0,C 180,E1 -12846.113,E2 -12846.113} C_VEL
LIN {X 0,Y 368.939,Z 404.528,A -85,B 0,C 180,E1 -12849.947,E2 -12849.947} C_VEL
LIN {X 0,Y 368.978,Z 404.521,A -85,B 0,C 180,E1 -12853.399,E2 -12853.399} C_VEL
LIN {X 0,Y 369.06,Z 404.514,A -85,B 0,C 180,E1 -12856.79,E2 -12856.79} C_VEL
LIN {X 0,Y 369.069,Z 404.513,A -85,B 0,C 180,E1 -12860.131,E2 -12860.131} C_VEL
LIN {X 0,Y 369.191,Z 404.5,A -85,B 0,C 180,E1 -12862.342,E2 -12862.342} C_VEL
LIN {X 0,Y 369.146,Z 404.504,A -85,B 0,C 180,E1 -12864.537,E2 -12864.537} C_VEL
LIN {X 0,Y 369.318,Z 404.481,A -85,B 0,C 180,E1 -12867.818,E2 -12867.818} C_VEL
LIN {X 0,Y 369.458,Z 404.465,A -85,B 0,C 180,E1 -12870,E2 -12870} C_VEL
LIN {X 0,Y 369.32,Z 404.484,A -85,B 0,C 180,E1 -12872.181,E2 -12872.181} C_VEL
LIN {X 0,Y 369.106,Z 404.508,A -85,B 0,C 180,E1 -12876.56,E2 -12876.56} C_VEL
LIN {X 0,Y 368.761,Z 404.551,A -85,B 0,C 180,E1 -12878.769,E2 -12878.769} C_VEL
LIN {X 0,Y 368.618,Z 405.047,A -85,B 0,C 180,E1 -12879.88,E2 -12879.88} C_VEL
LIN {X 0,Y 368.48,Z 408.914,A -85,B 0,C 180,E1 -12883.413,E2 -12883.413} C_VEL
LIN {X 0,Y 368.143,Z 413.333,A -85,B 0,C 180,E1 -12887.346,E2 -12887.346} C_VEL
LIN {X 0,Y 367.948,Z 417.124,A -85,B 0,C 180,E1 -12890.622,E2 -12890.622} C_VEL
LIN {X 0,Y 367.846,Z 420.81,A -85,B 0,C 180,E1 -12893.755,E2 -12893.755} C_VEL
LIN {X 0,Y 371.294,Z 435.639,A -85,B 0,C 180,E1 -12894.526,E2 -12894.526} C_VEL
LIN {X 0,Y 373.707,Z 447.973,A -85,B 0,C 180,E1 -12895.36,E2 -12895.36} C_VEL
LIN {X 0,Y 373.17,Z 458.201,A -85,B 0,C 180,E1 -12896.118,E2 -12896.118} C_VEL
LIN {X 0,Y 372.266,Z 469.501,A -85,B 0,C 180,E1 -12897.169,E2 -12897.169} C_VEL
LIN {X 0,Y 371.382,Z 479.975,A -85,B 0,C 180,E1 -12898.389,E2 -12898.389} C_VEL
LIN {X 0,Y 370.503,Z 489.194,A -85,B 0,C 180,E1 -12899.706,E2 -12899.706} C_VEL
LIN {X 0,Y 369.677,Z 497.61,A -85,B 0,C 180,E1 -12901.184,E2 -12901.184} C_VEL
LIN {X 0,Y 369.012,Z 504.328,A -85,B 0,C 180,E1 -12902.623,E2 -12902.623} C_VEL
LIN {X 0,Y 368.579,Z 509.016,A -85,B 0,C 180,E1 -12903.824,E2 -12903.824} C_VEL
LIN {X 0,Y 367.681,Z 511.843,A -85,B 0,C 180,E1 -12904.619,E2 -12904.619} C_VEL
LIN {X 0,Y 364.469,Z 515.925,A -85,B 0,C 180,E1 -12905.942,E2 -12905.942} C_VEL
LIN {X 0,Y 361.815,Z 518.655,A -85,B 0,C 180,E1 -12907.048,E2 -12907.048} C_VEL
LIN {X 0,Y 360.634,Z 520.441,A -85,B 0,C 180,E1 -12907.927,E2 -12907.927} C_VEL
LIN {X 0,Y 360.511,Z 520.941,A -85,B 0,C 180,E1 -12908.23,E2 -12908.23} C_VEL
LIN {X 0,Y 360.202,Z 523.902,A -85,B 0,C 180,E1 -12910.453,E2 -12910.453} C_VEL
LIN {X 0,Y 360.185,Z 525.036,A -85,B 0,C 180,E1 -12912.144,E2 -12912.144} C_VEL
LIN {X 0,Y 360.153,Z 525.268,A -85,B 0,C 180,E1 -12913.779,E2 -12913.779} C_VEL
LIN {X 0,Y 360.217,Z 524.678,A -85,B 0,C 180,E1 -12915.382,E2 -12915.382} C_VEL
LIN {X 0,Y 360.386,Z 523.308,A -85,B 0,C 180,E1 -12916.957,E2 -12916.957} C_VEL
LIN {X 0,Y 360.686,Z 521.126,A -85,B 0,C 180,E1 -12918.51,E2 -12918.51} C_VEL
LIN {X 0,Y 361.163,Z 516.851,A -85,B 0,C 180,E1 -12920.604,E2 -12920.604} C_VEL
LIN {X 0,Y 361.643,Z 512.5,A -85,B 0,C 180,E1 -12922.19,E2 -12922.19} C_VEL
LIN {X 0,Y 362.452,Z 505.807,A -85,B 0,C 180,E1 -12924.087,E2 -12924.087} C_VEL
LIN {X 0,Y 363.442,Z 497.71,A -85,B 0,C 180,E1 -12925.89,E2 -12925.89} C_VEL
LIN {X 0,Y 364.58,Z 488.567,A -85,B 0,C 180,E1 -12927.496,E2 -12927.496} C_VEL
LIN {X 0,Y 365.734,Z 478.935,A -85,B 0,C 180,E1 -12928.865,E2 -12928.865} C_VEL
LIN {X 0,Y 366.793,Z 468.972,A -85,B 0,C 180,E1 -12930.014,E2 -12930.014} C_VEL
LIN {X 0,Y 367.839,Z 457.587,A -85,B 0,C 180,E1 -12931.06,E2 -12931.06} C_VEL
LIN {X 0,Y 368.285,Z 451.786,A -85,B 0,C 180,E1 -12931.505,E2 -12931.505} C_VEL
LIN {X 0,Y 366.5,Z 442.054,A -85,B 0,C 180,E1 -12932.289,E2 -12932.289} C_VEL
LIN {X 0,Y 363.513,Z 430.46,A -85,B 0,C 180,E1 -12933.094,E2 -12933.094} C_VEL
LIN {X 0,Y 361.051,Z 422.329,A -85,B 0,C 180,E1 -12933.607,E2 -12933.607} C_VEL
LIN {X 0,Y 361.254,Z 418.644,A -85,B 0,C 180,E1 -12937.102,E2 -12937.102} C_VEL
LIN {X 0,Y 361.546,Z 414.954,A -85,B 0,C 180,E1 -12940.703,E2 -12940.703} C_VEL
LIN {X 0,Y 361.811,Z 411.489,A -85,B 0,C 180,E1 -12944.22,E2 -12944.22} C_VEL
LIN {X 0,Y 362.063,Z 409.304,A -85,B 0,C 180,E1 -12946.53,E2 -12946.53} C_VEL
LIN {X 0,Y 362.08,Z 406.233,A -85,B 0,C 180,E1 -12949.939,E2 -12949.939} C_VEL
LIN {X 0,Y 362.065,Z 405.392,A -85,B 0,C 180,E1 -12951.067,E2 -12951.067} C_VEL
LIN {X 0,Y 362.168,Z 405.375,A -85,B 0,C 180,E1 -12953.314,E2 -12953.314} C_VEL
LIN {X 0,Y 362.279,Z 405.362,A -85,B 0,C 180,E1 -12957.777,E2 -12957.777} C_VEL
LIN {X 0,Y 362.426,Z 405.342,A -85,B 0,C 180,E1 -12960,E2 -12960} C_VEL
LIN {X 0,Y 362.279,Z 405.357,A -85,B 0,C 180,E1 -12962.224,E2 -12962.224} C_VEL
LIN {X 0,Y 362.168,Z 405.374,A -85,B 0,C 180,E1 -12966.686,E2 -12966.686} C_VEL
LIN {X 0,Y 362.07,Z 405.387,A -85,B 0,C 180,E1 -12968.933,E2 -12968.933} C_VEL
LIN {X 0,Y 361.956,Z 405.401,A -85,B 0,C 180,E1 -12972.333,E2 -12972.333} C_VEL
LIN {X 0,Y 361.958,Z 405.399,A -85,B 0,C 180,E1 -12974.621,E2 -12974.621} C_VEL
LIN {X 0,Y 361.956,Z 405.4,A -85,B 0,C 180,E1 -12978.1,E2 -12978.1} C_VEL
LIN {X 0,Y 361.888,Z 405.409,A -85,B 0,C 180,E1 -12981.653,E2 -12981.653} C_VEL
LIN {X 0,Y 361.925,Z 405.404,A -85,B 0,C 180,E1 -12985.29,E2 -12985.29} C_VEL
LIN {X 0,Y 361.919,Z 405.405,A -85,B 0,C 180,E1 -12987.778,E2 -12987.778} C_VEL
LIN {X 0,Y 361.844,Z 405.414,A -85,B 0,C 180,E1 -12991.286,E2 -12991.286} C_VEL
LIN {X 0,Y 361.852,Z 405.414,A -85,B 0,C 180,E1 -12994.281,E2 -12994.281} C_VEL
LIN {X 0,Y 361.87,Z 405.413,A -85,B 0,C 180,E1 -12997.225,E2 -12997.225} C_VEL
LIN {X 0,Y 361.87,Z 405.413,A -85,B 0,C 180,E1 -13000.763,E2 -13000.763} C_VEL
LIN {X 0,Y 361.881,Z 405.516,A -85,B 0,C 180,E1 -13004.162,E2 -13004.162} C_VEL
LIN {X 0,Y 362.544,Z 409.347,A -85,B 0,C 180,E1 -13007.446,E2 -13007.446} C_VEL
LIN {X 0,Y 363.243,Z 413.563,A -85,B 0,C 180,E1 -13010.707,E2 -13010.707} C_VEL
LIN {X 0,Y 363.675,Z 417.078,A -85,B 0,C 180,E1 -13013.197,E2 -13013.197} C_VEL
LIN {X 0,Y 363.522,Z 421.246,A -85,B 0,C 180,E1 -13015.899,E2 -13015.899} C_VEL
LIN {X 0,Y 362.688,Z 427.618,A -85,B 0,C 180,E1 -13019.748,E2 -13019.748} C_VEL
LIN {X 0,Y 362.02,Z 434.136,A -85,B 0,C 180,E1 -13023.481,E2 -13023.481} C_VEL
LIN {X 0,Y 361.501,Z 440.756,A -85,B 0,C 180,E1 -13027.119,E2 -13027.119} C_VEL
LIN {X 0,Y 361.175,Z 445.069,A -85,B 0,C 180,E1 -13029.417,E2 -13029.417} C_VEL
LIN {X 0,Y 364.244,Z 459.153,A -85,B 0,C 180,E1 -13030.173,E2 -13030.173} C_VEL
LIN {X 0,Y 366.036,Z 470.851,A -85,B 0,C 180,E1 -13030.95,E2 -13030.95} C_VEL
LIN {X 0,Y 366.97,Z 482.882,A -85,B 0,C 180,E1 -13031.902,E2 -13031.902} C_VEL
LIN {X 0,Y 365.887,Z 494.69,A -85,B 0,C 180,E1 -13032.968,E2 -13032.968} C_VEL
LIN {X 0,Y 364.621,Z 505.515,A -85,B 0,C 180,E1 -13034.202,E2 -13034.202} C_VEL
LIN {X 0,Y 363.515,Z 516.19,A -85,B 0,C 180,E1 -13035.73,E2 -13035.73} C_VEL
LIN {X 0,Y 362.621,Z 524.107,A -85,B 0,C 180,E1 -13037.122,E2 -13037.122} C_VEL
LIN {X 0,Y 361.639,Z 531.871,A -85,B 0,C 180,E1 -13038.795,E2 -13038.795} C_VEL
LIN {X 0,Y 361.072,Z 538.136,A -85,B 0,C 180,E1 -13040.477,E2 -13040.477} C_VEL
LIN {X 0,Y 360.669,Z 543.134,A -85,B 0,C 180,E1 -13042.161,E2 -13042.161} C_VEL
LIN {X 0,Y 360.424,Z 547.251,A -85,B 0,C 180,E1 -13043.969,E2 -13043.969} C_VEL
LIN {X 0,Y 360.369,Z 549.856,A -85,B 0,C 180,E1 -13045.526,E2 -13045.526} C_VEL
LIN {X 0,Y 360.3,Z 552.169,A -85,B 0,C 180,E1 -13047.765,E2 -13047.765} C_VEL
LIN {X 0,Y 360.385,Z 552.713,A -85,B 0,C 180,E1 -13048.883,E2 -13048.883} C_VEL
LIN {X 0,Y 360.424,Z 552.822,A -85,B 0,C 180,E1 -13050,E2 -13050} C_VEL
LIN {X 0,Y 360.389,Z 552.536,A -85,B 0,C 180,E1 -13051.118,E2 -13051.118} C_VEL
LIN {X 0,Y 360.32,Z 551.856,A -85,B 0,C 180,E1 -13052.236,E2 -13052.236} C_VEL
LIN {X 0,Y 360.313,Z 550.756,A -85,B 0,C 180,E1 -13053.355,E2 -13053.355} C_VEL
LIN {X 0,Y 360.372,Z 549.206,A -85,B 0,C 180,E1 -13054.474,E2 -13054.474} C_VEL
LIN {X 0,Y 360.383,Z 546.489,A -85,B 0,C 180,E1 -13055.969,E2 -13055.969} C_VEL
LIN {X 0,Y 360.662,Z 541.855,A -85,B 0,C 180,E1 -13057.84,E2 -13057.84} C_VEL
LIN {X 0,Y 361.128,Z 535.428,A -85,B 0,C 180,E1 -13059.805,E2 -13059.805} C_VEL
LIN {X 0,Y 361.683,Z 528.403,A -85,B 0,C 180,E1 -13061.489,E2 -13061.489} C_VEL
LIN {X 0,Y 362.632,Z 519.61,A -85,B 0,C 180,E1 -13063.163,E2 -13063.163} C_VEL
LIN {X 0,Y 363.602,Z 509.542,A -85,B 0,C 180,E1 -13064.709,E2 -13064.709} C_VEL
LIN {X 0,Y 364.489,Z 499.473,A -85,B 0,C 180,E1 -13065.948,E2 -13065.948} C_VEL
LIN {X 0,Y 365.569,Z 488.27,A -85,B 0,C 180,E1 -13067.049,E2 -13067.049} C_VEL
LIN {X 0,Y 366.016,Z 481.541,A -85,B 0,C 180,E1 -13067.603,E2 -13067.603} C_VEL
LIN {X 0,Y 364.882,Z 470.269,A -85,B 0,C 180,E1 -13068.438,E2 -13068.438} C_VEL
LIN {X 0,Y 362.938,Z 457.116,A -85,B 0,C 180,E1 -13069.2,E2 -13069.2} C_VEL
LIN {X 0,Y 361.055,Z 446.285,A -85,B 0,C 180,E1 -13069.694,E2 -13069.694} C_VEL
LIN {X 0,Y 361.5,Z 439.165,A -85,B 0,C 180,E1 -13073.439,E2 -13073.439} C_VEL
LIN {X 0,Y 361.962,Z 433.039,A -85,B 0,C 180,E1 -13076.727,E2 -13076.727} C_VEL
LIN {X 0,Y 362.595,Z 426.608,A -85,B 0,C 180,E1 -13080.262,E2 -13080.262} C_VEL
LIN {X 0,Y 363.27,Z 419.794,A -85,B 0,C 180,E1 -13084.128,E2 -13084.128} C_VEL
LIN {X 0,Y 363.472,Z 417.113,A -85,B 0,C 180,E1 -13085.698,E2 -13085.698} C_VEL
LIN {X 0,Y 363.169,Z 412.918,A -85,B 0,C 180,E1 -13088.262,E2 -13088.262} C_VEL
LIN {X 0,Y 362.396,Z 408.312,A -85,B 0,C 180,E1 -13091.252,E2 -13091.252} C_VEL
LIN {X 0,Y 361.86,Z 405.413,A -85,B 0,C 180,E1 -13093.302,E2 -13093.302} C_VEL
LIN {X 0,Y 361.837,Z 405.416,A -85,B 0,C 180,E1 -13097.171,E2 -13097.171} C_VEL
LIN {X 0,Y 361.87,Z 405.41,A -85,B 0,C 180,E1 -13100.973,E2 -13100.973} C_VEL
LIN {X 0,Y 361.875,Z 405.407,A -85,B 0,C 180,E1 -13104.655,E2 -13104.655} C_VEL
LIN {X 0,Y 361.838,Z 405.411,A -85,B 0,C 180,E1 -13108.37,E2 -13108.37} C_VEL
LIN {X 0,Y 361.901,Z 405.407,A -85,B 0,C 180,E1 -13110.955,E2 -13110.955} C_VEL
LIN {X 0,Y 361.955,Z 405.399,A -85,B 0,C 180,E1 -13113.475,E2 -13113.475} C_VEL
LIN {X 0,Y 361.891,Z 405.409,A -85,B 0,C 180,E1 -13117.145,E2 -13117.145} C_VEL
LIN {X 0,Y 361.907,Z 405.405,A -85,B 0,C 180,E1 -13120.723,E2 -13120.723} C_VEL
LIN {X 0,Y 361.934,Z 405.404,A -85,B 0,C 180,E1 -13123.066,E2 -13123.066} C_VEL
LIN {X 0,Y 362,Z 405.392,A -85,B 0,C 180,E1 -13126.528,E2 -13126.528} C_VEL
LIN {X 0,Y 362.032,Z 405.386,A -85,B 0,C 180,E1 -13129.938,E2 -13129.938} C_VEL
LIN {X 0,Y 362.152,Z 405.372,A -85,B 0,C 180,E1 -13132.193,E2 -13132.193} C_VEL
LIN {X 0,Y 362.118,Z 405.377,A -85,B 0,C 180,E1 -13134.431,E2 -13134.431} C_VEL
LIN {X 0,Y 362.281,Z 405.356,A -85,B 0,C 180,E1 -13137.776,E2 -13137.776} C_VEL
LIN {X 0,Y 362.427,Z 405.337,A -85,B 0,C 180,E1 -13140,E2 -13140} C_VEL
LIN {X 0,Y 362.281,Z 405.356,A -85,B 0,C 180,E1 -13142.223,E2 -13142.223} C_VEL
LIN {X 0,Y 362.173,Z 405.373,A -85,B 0,C 180,E1 -13146.686,E2 -13146.686} C_VEL
LIN {X 0,Y 362.075,Z 405.386,A -85,B 0,C 180,E1 -13148.933,E2 -13148.933} C_VEL
LIN {X 0,Y 361.961,Z 405.397,A -85,B 0,C 180,E1 -13152.332,E2 -13152.332} C_VEL
LIN {X 0,Y 361.963,Z 405.399,A -85,B 0,C 180,E1 -13154.62,E2 -13154.62} C_VEL
LIN {X 0,Y 361.96,Z 405.396,A -85,B 0,C 180,E1 -13158.099,E2 -13158.099} C_VEL
LIN {X 0,Y 361.893,Z 405.404,A -85,B 0,C 180,E1 -13161.653,E2 -13161.653} C_VEL
LIN {X 0,Y 361.929,Z 405.4,A -85,B 0,C 180,E1 -13165.29,E2 -13165.29} C_VEL
LIN {X 0,Y 361.919,Z 405.4,A -85,B 0,C 180,E1 -13167.778,E2 -13167.778} C_VEL
LIN {X 0,Y 361.847,Z 405.41,A -85,B 0,C 180,E1 -13171.285,E2 -13171.285} C_VEL
LIN {X 0,Y 361.855,Z 405.411,A -85,B 0,C 180,E1 -13174.28,E2 -13174.28} C_VEL
LIN {X 0,Y 361.864,Z 405.408,A -85,B 0,C 180,E1 -13177.223,E2 -13177.223} C_VEL
LIN {X 0,Y 361.836,Z 405.415,A -85,B 0,C 180,E1 -13180.755,E2 -13180.755} C_VEL
LIN {X 0,Y 361.818,Z 405.416,A -85,B 0,C 180,E1 -13184.368,E2 -13184.368} C_VEL
LIN {X 0,Y 361.837,Z 405.411,A -85,B 0,C 180,E1 -13187.568,E2 -13187.568} C_VEL
LIN {X 0,Y 361.872,Z 405.409,A -85,B 0,C 180,E1 -13190.973,E2 -13190.973} C_VEL
LIN {X 0,Y 361.876,Z 405.411,A -85,B 0,C 180,E1 -13194.655,E2 -13194.655} C_VEL
LIN {X 0,Y 361.839,Z 405.415,A -85,B 0,C 180,E1 -13198.371,E2 -13198.371} C_VEL
LIN {X 0,Y 361.91,Z 405.405,A -85,B 0,C 180,E1 -13202.221,E2 -13202.221} C_VEL
LIN {X 0,Y 361.93,Z 405.403,A -85,B 0,C 180,E1 -13204.71,E2 -13204.71} C_VEL
LIN {X 0,Y 361.894,Z 405.409,A -85,B 0,C 180,E1 -13208.347,E2 -13208.347} C_VEL
LIN {X 0,Y 361.969,Z 405.397,A -85,B 0,C 180,E1 -13212.061,E2 -13212.061} C_VEL
LIN {X 0,Y 362,Z 405.394,A -85,B 0,C 180,E1 -13216.101,E2 -13216.101} C_VEL
LIN {X 0,Y 362.033,Z 405.388,A -85,B 0,C 180,E1 -13219.938,E2 -13219.938} C_VEL
LIN {X 0,Y 362.149,Z 405.376,A -85,B 0,C 180,E1 -13222.192,E2 -13222.192} C_VEL
LIN {X 0,Y 362.12,Z 405.381,A -85,B 0,C 180,E1 -13224.431,E2 -13224.431} C_VEL
LIN {X 0,Y 362.282,Z 405.357,A -85,B 0,C 180,E1 -13227.776,E2 -13227.776} C_VEL
LIN {X 0,Y 362.428,Z 405.34,A -85,B 0,C 180,E1 -13230,E2 -13230} C_VEL
LIN {X 0,Y 362.284,Z 405.36,A -85,B 0,C 180,E1 -13232.223,E2 -13232.223} C_VEL
LIN {X 0,Y 362.056,Z 405.385,A -85,B 0,C 180,E1 -13236.688,E2 -13236.688} C_VEL
LIN {X 0,Y 361.672,Z 405.434,A -85,B 0,C 180,E1 -13238.943,E2 -13238.943} C_VEL
LIN {X 0,Y 361.562,Z 406.133,A -85,B 0,C 180,E1 -13240.075,E2 -13240.075} C_VEL
LIN {X 0,Y 361.416,Z 409.842,A -85,B 0,C 180,E1 -13243.52,E2 -13243.52} C_VEL
LIN {X 0,Y 361.08,Z 414.281,A -85,B 0,C 180,E1 -13247.498,E2 -13247.498} C_VEL
LIN {X 0,Y 360.853,Z 417.996,A -85,B 0,C 180,E1 -13250.796,E2 -13250.796} C_VEL
LIN {X 0,Y 360.798,Z 421.234,A -85,B 0,C 180,E1 -13253.43,E2 -13253.43} C_VEL
LIN {X 0,Y 363.905,Z 434.419,A -85,B 0,C 180,E1 -13254.11,E2 -13254.11} C_VEL
LIN {X 0,Y 366.469,Z 446.914,A -85,B 0,C 180,E1 -13254.954,E2 -13254.954} C_VEL
LIN {X 0,Y 366.838,Z 451.612,A -85,B 0,C 180,E1 -13255.307,E2 -13255.307} C_VEL
LIN {X 0,Y 365.96,Z 462.784,A -85,B 0,C 180,E1 -13256.212,E2 -13256.212} C_VEL
LIN {X 0,Y 365.04,Z 473.915,A -85,B 0,C 180,E1 -13257.364,E2 -13257.364} C_VEL
LIN {X 0,Y 364.012,Z 484.284,A -85,B 0,C 180,E1 -13258.702,E2 -13258.702} C_VEL
LIN {X 0,Y 363.132,Z 493.722,A -85,B 0,C 180,E1 -13260.211,E2 -13260.211} C_VEL
LIN {X 0,Y 362.215,Z 502.249,A -85,B 0,C 180,E1 -13261.919,E2 -13261.919} C_VEL
LIN {X 0,Y 361.511,Z 509.657,A -85,B 0,C 180,E1 -13263.787,E2 -13263.787} C_VEL
LIN {X 0,Y 360.963,Z 515.585,A -85,B 0,C 180,E1 -13265.739,E2 -13265.739} C_VEL
LIN {X 0,Y 360.674,Z 518.958,A -85,B 0,C 180,E1 -13267.16,E2 -13267.16} C_VEL
LIN {X 0,Y 360.511,Z 520.941,A -85,B 0,C 180,E1 -13268.23,E2 -13268.23} C_VEL
LIN {X 0,Y 359.741,Z 522.39,A -85,B 0,C 180,E1 -13269.133,E2 -13269.133} C_VEL
LIN {X 0,Y 356.737,Z 524.206,A -85,B 0,C 180,E1 -13270.615,E2 -13270.615} C_VEL
LIN {X 0,Y 354.234,Z 525.122,A -85,B 0,C 180,E1 -13271.826,E2 -13271.826} C_VEL
LIN {X 0,Y 353.154,Z 525.49,A -85,B 0,C 180,E1 -13272.771,E2 -13272.771} C_VEL
LIN {X 0,Y 353.061,Z 525.477,A -85,B 0,C 180,E1 -13273.092,E2 -13273.092} C_VEL
LIN {X 0,Y 353.083,Z 525.501,A -85,B 0,C 180,E1 -13274.228,E2 -13274.228} C_VEL
LIN {X 0,Y 353.175,Z 524.701,A -85,B 0,C 180,E1 -13275.855,E2 -13275.855} C_VEL
LIN {X 0,Y 353.374,Z 523.129,A -85,B 0,C 180,E1 -13277.452,E2 -13277.452} C_VEL
LIN {X 0,Y 353.907,Z 519.333,A -85,B 0,C 180,E1 -13279.805,E2 -13279.805} C_VEL
LIN {X 0,Y 354.297,Z 515.662,A -85,B 0,C 180,E1 -13281.399,E2 -13281.399} C_VEL
LIN {X 0,Y 354.929,Z 510.919,A -85,B 0,C 180,E1 -13283.011,E2 -13283.011} C_VEL
LIN {X 0,Y 355.665,Z 505.056,A -85,B 0,C 180,E1 -13284.617,E2 -13284.617} C_VEL
LIN {X 0,Y 356.607,Z 497.803,A -85,B 0,C 180,E1 -13286.223,E2 -13286.223} C_VEL
LIN {X 0,Y 357.643,Z 489.824,A -85,B 0,C 180,E1 -13287.669,E2 -13287.669} C_VEL
LIN {X 0,Y 358.83,Z 480.424,A -85,B 0,C 180,E1 -13289.061,E2 -13289.061} C_VEL
LIN {X 0,Y 360.026,Z 470.05,A -85,B 0,C 180,E1 -13290.308,E2 -13290.308} C_VEL
LIN {X 0,Y 361.108,Z 459.061,A -85,B 0,C 180,E1 -13291.363,E2 -13291.363} C_VEL
LIN {X 0,Y 361.567,Z 452.619,A -85,B 0,C 180,E1 -13291.877,E2 -13291.877} C_VEL
LIN {X 0,Y 359.176,Z 440.455,A -85,B 0,C 180,E1 -13292.88,E2 -13292.88} C_VEL
LIN {X 0,Y 355.935,Z 429.013,A -85,B 0,C 180,E1 -13293.691,E2 -13293.691} C_VEL
LIN {X 0,Y 354.051,Z 422.643,A -85,B 0,C 180,E1 -13294.106,E2 -13294.106} C_VEL
LIN {X 0,Y 354.253,Z 418.776,A -85,B 0,C 180,E1 -13297.856,E2 -13297.856} C_VEL
LIN {X 0,Y 354.471,Z 416.327,A -85,B 0,C 180,E1 -13300.303,E2 -13300.303} C_VEL
LIN {X 0,Y 354.745,Z 412.849,A -85,B 0,C 180,E1 -13303.897,E2 -13303.897} C_VEL
LIN {X 0,Y 355.044,Z 410.635,A -85,B 0,C 180,E1 -13306.259,E2 -13306.259} C_VEL
LIN {X 0,Y 355.068,Z 407.571,A -85,B 0,C 180,E1 -13309.739,E2 -13309.739} C_VEL
LIN {X 0,Y 355.119,Z 406.256,A -85,B 0,C 180,E1 -13311.695,E2 -13311.695} C_VEL
LIN {X 0,Y 355.089,Z 406.256,A -85,B 0,C 180,E1 -13314.321,E2 -13314.321} C_VEL
LIN {X 0,Y 355.242,Z 406.238,A -85,B 0,C 180,E1 -13317.732,E2 -13317.732} C_VEL
LIN {X 0,Y 355.395,Z 406.218,A -85,B 0,C 180,E1 -13320,E2 -13320} C_VEL
LIN {X 0,Y 355.242,Z 406.233,A -85,B 0,C 180,E1 -13322.268,E2 -13322.268} C_VEL
LIN {X 0,Y 355.134,Z 406.25,A -85,B 0,C 180,E1 -13326.819,E2 -13326.819} C_VEL
LIN {X 0,Y 355.011,Z 406.265,A -85,B 0,C 180,E1 -13329.113,E2 -13329.113} C_VEL
LIN {X 0,Y 354.917,Z 406.277,A -85,B 0,C 180,E1 -13332.581,E2 -13332.581} C_VEL
LIN {X 0,Y 354.886,Z 406.28,A -85,B 0,C 180,E1 -13336.096,E2 -13336.096} C_VEL
LIN {X 0,Y 354.902,Z 406.278,A -85,B 0,C 180,E1 -13338.472,E2 -13338.472} C_VEL
LIN {X 0,Y 354.831,Z 406.287,A -85,B 0,C 180,E1 -13342.106,E2 -13342.106} C_VEL
LIN {X 0,Y 354.896,Z 406.279,A -85,B 0,C 180,E1 -13345.828,E2 -13345.828} C_VEL
LIN {X 0,Y 354.851,Z 406.285,A -85,B 0,C 180,E1 -13349.679,E2 -13349.679} C_VEL
LIN {X 0,Y 354.803,Z 406.292,A -85,B 0,C 180,E1 -13353.703,E2 -13353.703} C_VEL
LIN {X 0,Y 354.799,Z 406.294,A -85,B 0,C 180,E1 -13356.459,E2 -13356.459} C_VEL
LIN {X 0,Y 354.821,Z 406.293,A -85,B 0,C 180,E1 -13359.424,E2 -13359.424} C_VEL
LIN {X 0,Y 354.804,Z 406.292,A -85,B 0,C 180,E1 -13362.871,E2 -13362.871} C_VEL
LIN {X 0,Y 354.822,Z 406.426,A -85,B 0,C 180,E1 -13363.608,E2 -13363.608} C_VEL
LIN {X 0,Y 355.507,Z 410.254,A -85,B 0,C 180,E1 -13367.009,E2 -13367.009} C_VEL
LIN {X 0,Y 356.192,Z 414.375,A -85,B 0,C 180,E1 -13370.31,E2 -13370.31} C_VEL
LIN {X 0,Y 356.677,Z 418.123,A -85,B 0,C 180,E1 -13373.061,E2 -13373.061} C_VEL
LIN {X 0,Y 356.489,Z 422.387,A -85,B 0,C 180,E1 -13375.895,E2 -13375.895} C_VEL
LIN {X 0,Y 355.648,Z 428.615,A -85,B 0,C 180,E1 -13379.742,E2 -13379.742} C_VEL
LIN {X 0,Y 354.957,Z 435.159,A -85,B 0,C 180,E1 -13383.575,E2 -13383.575} C_VEL
LIN {X 0,Y 354.422,Z 441.727,A -85,B 0,C 180,E1 -13387.253,E2 -13387.253} C_VEL
LIN {X 0,Y 354.164,Z 444.785,A -85,B 0,C 180,E1 -13388.932,E2 -13388.932} C_VEL
LIN {X 0,Y 357.224,Z 458.368,A -85,B 0,C 180,E1 -13389.676,E2 -13389.676} C_VEL
LIN {X 0,Y 359.307,Z 471.44,A -85,B 0,C 180,E1 -13390.579,E2 -13390.579} C_VEL
LIN {X 0,Y 360.196,Z 483.288,A -85,B 0,C 180,E1 -13391.554,E2 -13391.554} C_VEL
LIN {X 0,Y 359.233,Z 493.486,A -85,B 0,C 180,E1 -13392.495,E2 -13392.495} C_VEL
LIN {X 0,Y 357.916,Z 504.501,A -85,B 0,C 180,E1 -13393.752,E2 -13393.752} C_VEL
